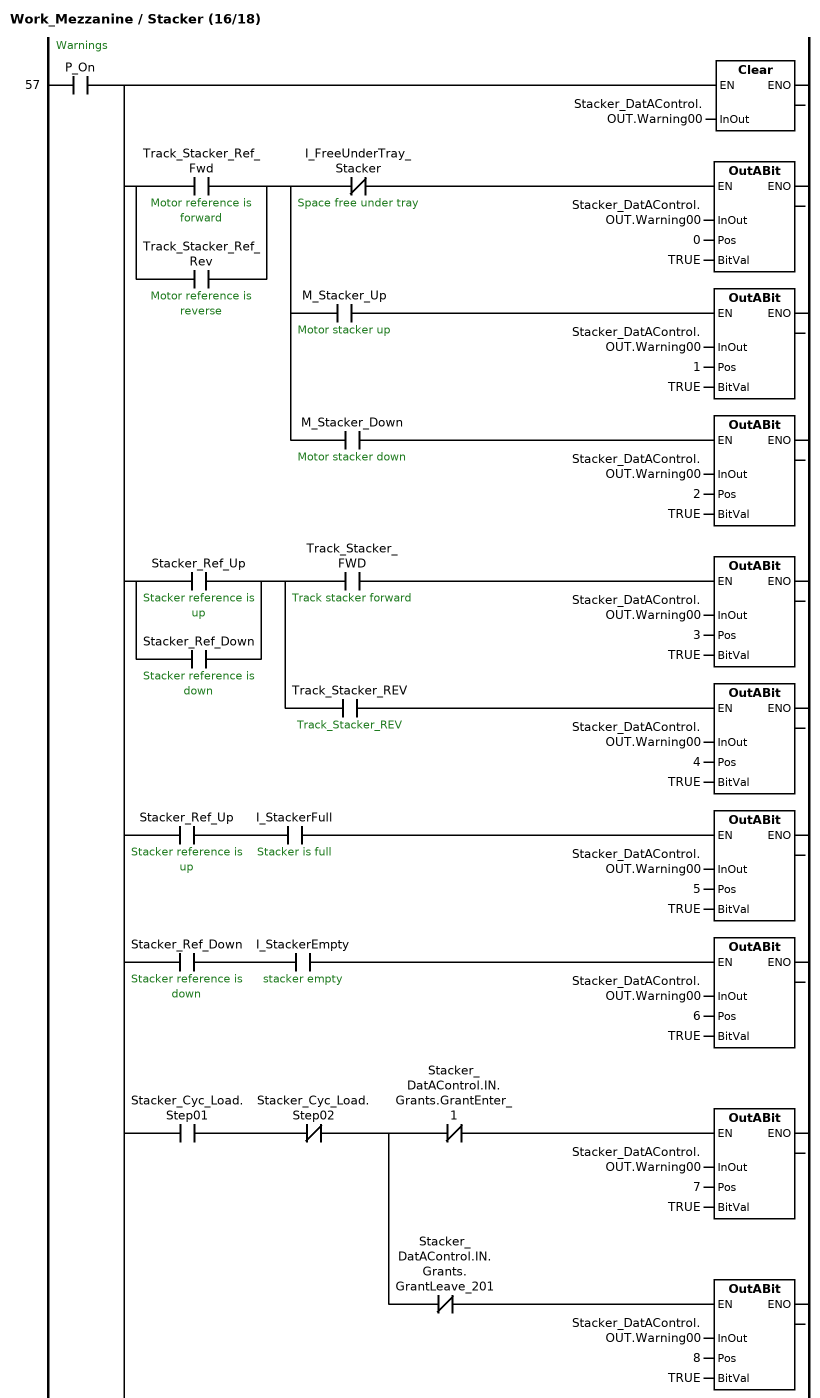
(* [picture p126: Work_Mezzanine / Stacker, rungs 57-57] *)

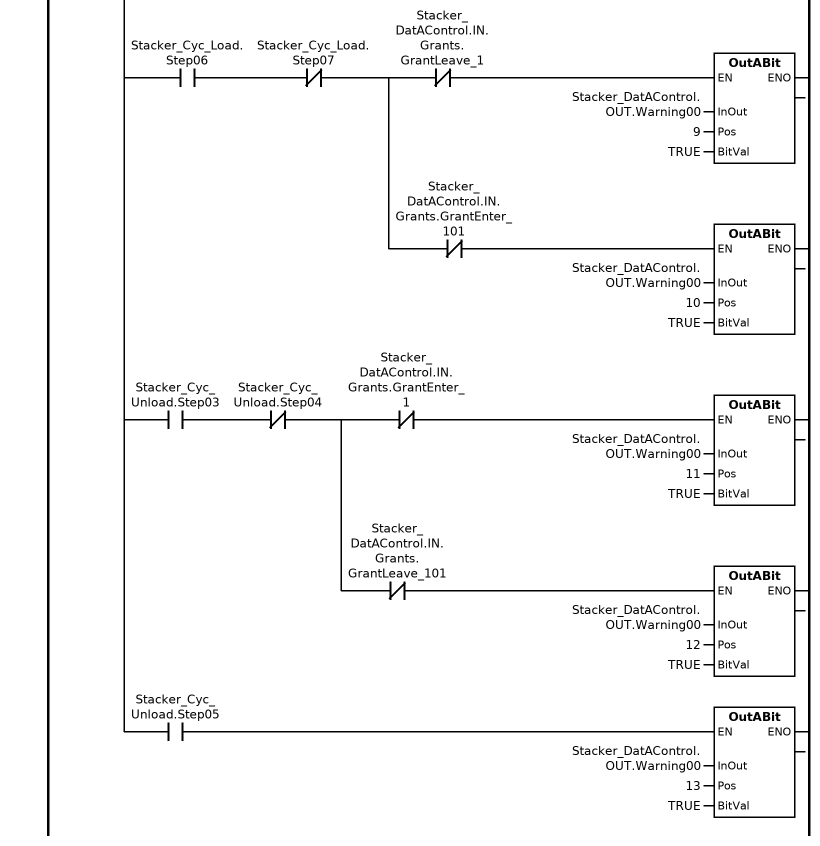
(* Rung 57: Warnings *)
IF P_On THEN Clear(InOut := Stacker_DatAControl.OUT.Warning00); END_IF;
_p6 := P_On AND (Track_Stacker_Ref_Fwd OR Track_Stacker_Ref_Rev);
IF _p6 AND NOT I_FreeUnderTray_Stacker THEN
    OutABit(InOut := Stacker_DatAControl.OUT.Warning00, Pos := 0, BitVal := TRUE);
END_IF;
IF _p6 AND M_Stacker_Up THEN
    OutABit(InOut := Stacker_DatAControl.OUT.Warning00, Pos := 1, BitVal := TRUE);
END_IF;
IF _p6 AND M_Stacker_Down THEN
    OutABit(InOut := Stacker_DatAControl.OUT.Warning00, Pos := 2, BitVal := TRUE);
END_IF;
IF P_On AND (Stacker_Ref_Up OR Stacker_Ref_Down) AND Track_Stacker_FWD THEN
    OutABit(InOut := Stacker_DatAControl.OUT.Warning00, Pos := 3, BitVal := TRUE);
END_IF;
IF P_On AND (Stacker_Ref_Up OR Stacker_Ref_Down) AND Track_Stacker_REV THEN
    OutABit(InOut := Stacker_DatAControl.OUT.Warning00, Pos := 4, BitVal := TRUE);
END_IF;
IF P_On AND Stacker_Ref_Up AND I_StackerFull THEN
    OutABit(InOut := Stacker_DatAControl.OUT.Warning00, Pos := 5, BitVal := TRUE);
END_IF;
IF P_On AND Stacker_Ref_Down AND I_StackerEmpty THEN
    OutABit(InOut := Stacker_DatAControl.OUT.Warning00, Pos := 6, BitVal := TRUE);
END_IF;
_p7 := P_On AND Stacker_Cyc_Load.Step01 AND NOT Stacker_Cyc_Load.Step02;
IF _p7 AND NOT Stacker_DatAControl.IN.Grants.GrantEnter_1 THEN
    OutABit(InOut := Stacker_DatAControl.OUT.Warning00, Pos := 7, BitVal := TRUE);
END_IF;
IF _p7 AND NOT Stacker_DatAControl.IN.Grants.GrantLeave_201 THEN
    OutABit(InOut := Stacker_DatAControl.OUT.Warning00, Pos := 8, BitVal := TRUE);
END_IF;
_p8 := P_On AND Stacker_Cyc_Load.Step06 AND NOT Stacker_Cyc_Load.Step07;
IF _p8 AND NOT Stacker_DatAControl.IN.Grants.GrantLeave_1 THEN
    OutABit(InOut := Stacker_DatAControl.OUT.Warning00, Pos := 9, BitVal := TRUE);
END_IF;
IF _p8 AND NOT Stacker_DatAControl.IN.Grants.GrantEnter_101 THEN
    OutABit(InOut := Stacker_DatAControl.OUT.Warning00, Pos := 10, BitVal := TRUE);
END_IF;
_p9 := P_On AND Stacker_Cyc_Unload.Step03 AND NOT Stacker_Cyc_Unload.Step04;
IF _p9 AND NOT Stacker_DatAControl.IN.Grants.GrantEnter_1 THEN
    OutABit(InOut := Stacker_DatAControl.OUT.Warning00, Pos := 11, BitVal := TRUE);
END_IF;
IF _p9 AND NOT Stacker_DatAControl.IN.Grants.GrantLeave_101 THEN
    OutABit(InOut := Stacker_DatAControl.OUT.Warning00, Pos := 12, BitVal := TRUE);
END_IF;
IF P_On AND Stacker_Cyc_Unload.Step05 THEN
    OutABit(InOut := Stacker_DatAControl.OUT.Warning00, Pos := 13, BitVal := TRUE);
END_IF;

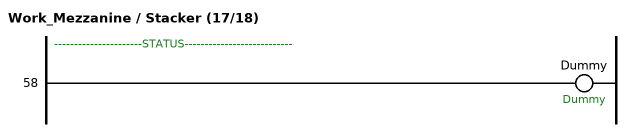
(* Rung 58: ----------------------STATUS--------------------------- *)
Dummy := TRUE;

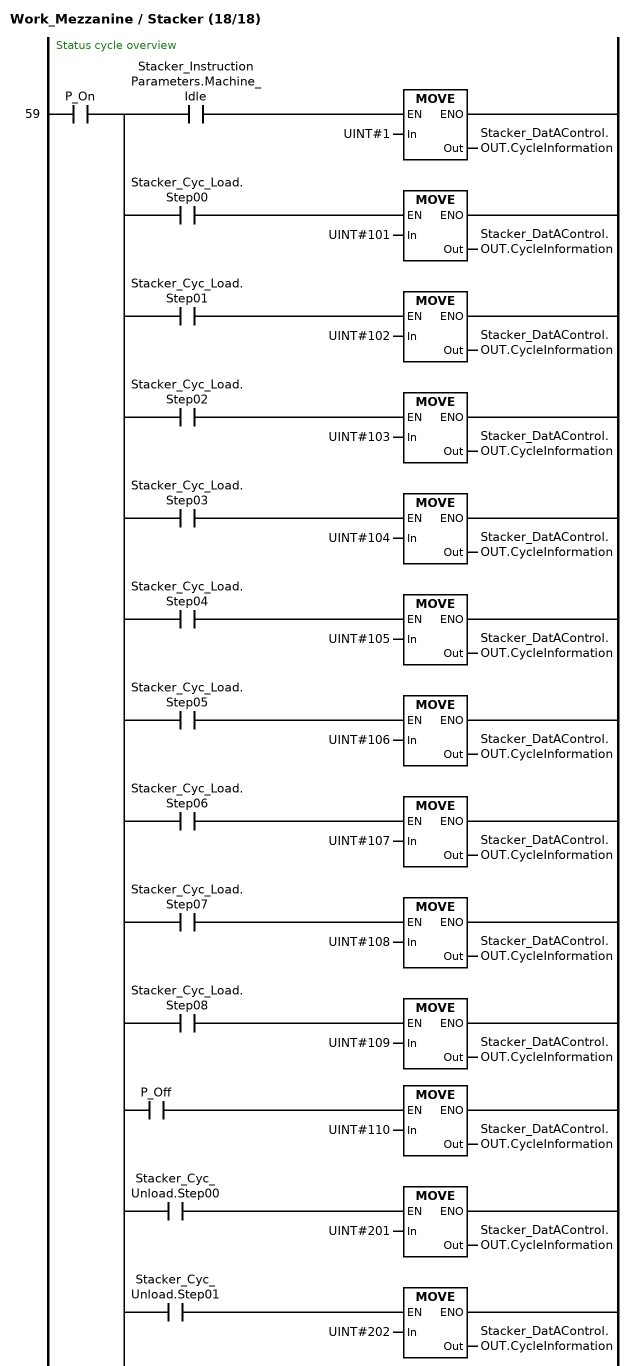

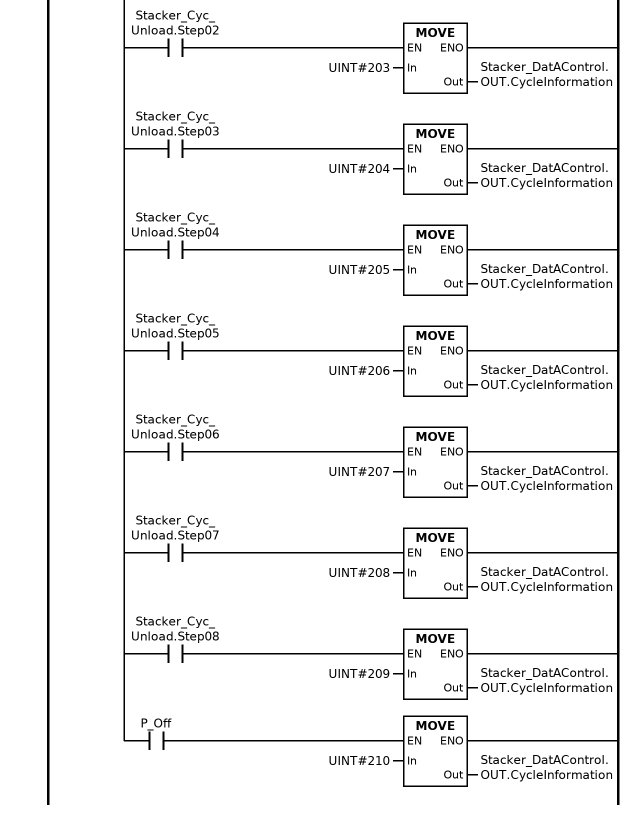
(* Rung 59: Status cycle overview *)
IF P_On AND Stacker_InstructionParameters.Machine_Idle THEN
    Stacker_DatAControl.OUT.CycleInformation := UINT#1;
END_IF;
IF P_On AND Stacker_Cyc_Load.Step00 THEN Stacker_DatAControl.OUT.CycleInformation := UINT#101; END_IF;
IF P_On AND Stacker_Cyc_Load.Step01 THEN Stacker_DatAControl.OUT.CycleInformation := UINT#102; END_IF;
IF P_On AND Stacker_Cyc_Load.Step02 THEN Stacker_DatAControl.OUT.CycleInformation := UINT#103; END_IF;
IF P_On AND Stacker_Cyc_Load.Step03 THEN Stacker_DatAControl.OUT.CycleInformation := UINT#104; END_IF;
IF P_On AND Stacker_Cyc_Load.Step04 THEN Stacker_DatAControl.OUT.CycleInformation := UINT#105; END_IF;
IF P_On AND Stacker_Cyc_Load.Step05 THEN Stacker_DatAControl.OUT.CycleInformation := UINT#106; END_IF;
IF P_On AND Stacker_Cyc_Load.Step06 THEN Stacker_DatAControl.OUT.CycleInformation := UINT#107; END_IF;
IF P_On AND Stacker_Cyc_Load.Step07 THEN Stacker_DatAControl.OUT.CycleInformation := UINT#108; END_IF;
IF P_On AND Stacker_Cyc_Load.Step08 THEN Stacker_DatAControl.OUT.CycleInformation := UINT#109; END_IF;
IF P_On AND P_Off THEN Stacker_DatAControl.OUT.CycleInformation := UINT#110; END_IF;
IF P_On AND Stacker_Cyc_Unload.Step00 THEN Stacker_DatAControl.OUT.CycleInformation := UINT#201; END_IF;
IF P_On AND Stacker_Cyc_Unload.Step01 THEN Stacker_DatAControl.OUT.CycleInformation := UINT#202; END_IF;
IF P_On AND Stacker_Cyc_Unload.Step02 THEN Stacker_DatAControl.OUT.CycleInformation := UINT#203; END_IF;
IF P_On AND Stacker_Cyc_Unload.Step03 THEN Stacker_DatAControl.OUT.CycleInformation := UINT#204; END_IF;
IF P_On AND Stacker_Cyc_Unload.Step04 THEN Stacker_DatAControl.OUT.CycleInformation := UINT#205; END_IF;
IF P_On AND Stacker_Cyc_Unload.Step05 THEN Stacker_DatAControl.OUT.CycleInformation := UINT#206; END_IF;
IF P_On AND Stacker_Cyc_Unload.Step06 THEN Stacker_DatAControl.OUT.CycleInformation := UINT#207; END_IF;
IF P_On AND Stacker_Cyc_Unload.Step07 THEN Stacker_DatAControl.OUT.CycleInformation := UINT#208; END_IF;
IF P_On AND Stacker_Cyc_Unload.Step08 THEN Stacker_DatAControl.OUT.CycleInformation := UINT#209; END_IF;
IF P_On AND P_Off THEN Stacker_DatAControl.OUT.CycleInformation := UINT#210; END_IF;
END_PROGRAM

PROGRAM ReadSettings
VAR_EXTERNAL
    Dummy : BOOL;
    Settings_CP : ST_Settings_CP;
    XTrack_X_Values : ARRAY[0..49] OF UDINT;
    XTrack_Y_Values : ARRAY[0..49] OF UDINT;
    Area : ARRAY[0..99] OF ST_Area;
    XTrack : ARRAY[0..49] OF ST_XTrack;
    Lift : ARRAY[0..9] OF ST_LiftInformation;
END_VAR
// Margins reservation system.
Settings_CP.Setting_Margin_X:= 1350; // Minimum margin = pallet 1200/2. 1270
Settings_CP.Setting_Margin_Y:= 700; // Minimum margin = Carrier lenght/2.

// Margin to define if carrier is in a certain area.
Settings_CP.Margin_AreaCompare:= 100;

// Values of position in X direction
XTrack_X_Values[0]:= 0;
XTrack_X_Values[1]:= 100000;
XTrack_X_Values[2]:= 102800;
XTrack_X_Values[3]:= 105600;
XTrack_X_Values[4]:= 108400;
XTrack_X_Values[5]:= 111516;
XTrack_X_Values[6]:= 114316;
XTrack_X_Values[7]:= 117116;
XTrack_X_Values[8]:= 119916;
XTrack_X_Values[9]:= 122716;
XTrack_X_Values[10]:= 125928;
XTrack_X_Values[11]:= 128728;
XTrack_X_Values[12]:= 131528;
XTrack_X_Values[13]:= 134328;
XTrack_X_Values[14]:= 137128;
XTrack_X_Values[15]:= 140244;
XTrack_X_Values[16]:= 143044;
XTrack_X_Values[17]:= 145844;
XTrack_X_Values[18]:= 148644;
XTrack_X_Values[19]:= 151444;

// Values of positions X-Track in Y direction
XTrack_Y_Values[0]:= 0;
XTrack_Y_Values[1]:= 100000;
XTrack_Y_Values[2]:= 108098;

// Dimensions of areas
// Check electrical lay-out for and overview of the Areas.

// This area is always 0
Area[0].Level:= 0;
Area[0].X_MIN:= 0;
Area[0].X_MAX:= 0;
Area[0].Y_Back:= 0;
Area[0].Y_Front:= 0;

// This is the 1st area on level 1, see lay-out for details.
// 1 to 9 = 100000 - 1/2 carrier with(650) to 122716 + 1/2 carrier with(650)
Area[11].Level:= 1;
Area[11].X_MIN:= 99350;
Area[11].X_MAX:= 123366;
Area[11].Y_Back:= 105198;
Area[11].Y_Front:= 110998;

// This is the 2nd area on level 1, see lay-out for details.
// 1 to 9
Area[12].Level:= 1;
Area[12].X_MIN:= 99350;
Area[12].X_MAX:= 123366;
Area[12].Y_Back:= 97100;
Area[12].Y_Front:= 102900; //carrier hit end @12981

// This is the 3th area on level 1, see lay-out for details.
// 10
Area[13].Level:= 1;
Area[13].X_MIN:= 125278;
Area[13].X_MAX:= 126578;
Area[13].Y_Back:= 98200;
Area[13].Y_Front:= 110998;

// This is the 4th area on level 1, see lay-out for details.
//1 to 19
Area[14].Level:= 1;
Area[14].X_MIN:= 128078;
Area[14].X_MAX:= 152094;
Area[14].Y_Back:= 105198;
Area[14].Y_Front:= 110998;

// This is the 5th area on level 1, see lay-out for details.
// 11 to 16
Area[15].Level:= 1;
Area[15].X_MIN:= 128078;
Area[15].X_MAX:= 143694;
Area[15].Y_Back:= 97100;
Area[15].Y_Front:= 102900;

// This is the 6th area on level 1, see lay-out for details.
// 17
Area[16].Level:= 1;
Area[16].X_MIN:= 145194;
Area[16].X_MAX:= 146494;
Area[16].Y_Back:= 98200;
Area[16].Y_Front:= 102900;

// This is the 7th area on level 1, see lay-out for details.
// 18 to 19
Area[17].Level:= 1;
Area[17].X_MIN:= 147994;
Area[17].X_MAX:= 152094;
Area[17].Y_Back:= 97100;
Area[17].Y_Front:= 102900;

// Copy areas to other levels
Area[21]:= Area[11];
Area[21].Level:= 2;
Area[31]:= Area[11];
Area[31].Level:= 3;
Area[41]:= Area[11];
Area[41].Level:= 4;
Area[51]:= Area[11];
Area[51].Level:= 5;
Area[61]:= Area[11];
Area[61].Level:= 6;
Area[71]:= Area[11];
Area[71].Level:= 7;

Area[22]:= Area[12];
Area[22].Level:= 2;
Area[32]:= Area[12];
Area[32].Level:= 3;
Area[42]:= Area[12];
Area[42].Level:= 4;
Area[52]:= Area[12];
Area[52].Level:= 5;
Area[62]:= Area[12];
Area[62].Level:= 6;
Area[72]:= Area[12];
Area[72].Level:= 7;

Area[23]:= Area[13];
Area[23].Level:= 2;
Area[33]:= Area[13];
Area[33].Level:= 3;
Area[43]:= Area[13];
Area[43].Level:= 4;
Area[53]:= Area[13];
Area[53].Level:= 5;
Area[63]:= Area[13];
Area[63].Level:= 6;
Area[73]:= Area[13];
Area[73].Level:= 7;

Area[24]:= Area[14];
Area[24].Level:= 2;
Area[34]:= Area[14];
Area[34].Level:= 3;
Area[44]:= Area[14];
Area[44].Level:= 4;
Area[54]:= Area[14];
Area[54].Level:= 5;
Area[64]:= Area[14];
Area[64].Level:= 6;
Area[74]:= Area[14];
Area[74].Level:= 7;

Area[25]:= Area[15];
Area[25].Level:= 2;
Area[35]:= Area[15];
Area[35].Level:= 3;
Area[45]:= Area[15];
Area[45].Level:= 4;
Area[55]:= Area[15];
Area[55].Level:= 5;
Area[65]:= Area[15];
Area[65].Level:= 6;
Area[75]:= Area[15];
Area[75].Level:= 7;

Area[26]:= Area[16];
Area[26].Level:= 2;
Area[36]:= Area[16];
Area[36].Level:= 3;
Area[46]:= Area[16];
Area[46].Level:= 4;
Area[56]:= Area[16];
Area[56].Level:= 5;
Area[66]:= Area[16];
Area[66].Level:= 6;
Area[76]:= Area[16];
Area[76].Level:= 7;

Area[27]:= Area[17];
Area[27].Level:= 2;
Area[37]:= Area[17];
Area[37].Level:= 3;
Area[47]:= Area[17];
Area[47].Level:= 4;
Area[57]:= Area[17];
Area[57].Level:= 5;
Area[67]:= Area[17];
Area[67].Level:= 6;
Area[77]:= Area[17];
Area[77].Level:= 7;

 // Information about X-Tracks
XTrack[0].XTrack_Number:= 0;
XTrack[0].MinimumPosition:= 0;
XTrack[0].MaximumPosition:= 0;
	 
XTrack[1].XTrack_Number:= 1;
XTrack[1].MinimumPosition:= 1;
XTrack[1].MaximumPosition:= 19;

XTrack[2].XTrack_Number:= 2;
XTrack[2].MinimumPosition:= 1;
XTrack[2].MaximumPosition:= 19;

// Information about lifts
// This lift is always 0
Lift[0].Number:= 0;
Lift[0].X_Coordinate_Lift_MIN:= 0;
Lift[0].X_Coordinate_Lift_MAX:= 0;
Lift[0].Y_Coordinate_Lift_Back:= 0;
Lift[0].Y_Coordinate_Lift_Front:= 0;
Lift[0].Y_Coordinate_LiftCenter:= 0;
Lift[0].Pos_Lift_XTrack:= FALSE;

// This is the lift in growing room3
Lift[1].Number:= 1;
Lift[1].X_Coordinate_Lift_MIN:= 125278;
Lift[1].X_Coordinate_Lift_MAX:= 126578;
Lift[1].Y_Coordinate_Lift_Back:= 98100;
Lift[1].Y_Coordinate_Lift_Front:= 99390;
Lift[1].Y_Coordinate_LiftCenter:= 98223; 
Lift[1].Pos_Lift_XTrack:= FALSE;

// This is the lift in growing room4 ;
Lift[2].Number:= 2;
Lift[2].X_Coordinate_Lift_MIN:= 145194;
Lift[2].X_Coordinate_Lift_MAX:= 146494;
Lift[2].Y_Coordinate_Lift_Back:= 98100;
Lift[2].Y_Coordinate_Lift_Front:= 99390;
Lift[2].Y_Coordinate_LiftCenter:= 98223;
Lift[2].Pos_Lift_XTrack:= FALSE;
END_PROGRAM

FUNCTION PositionResetCheck : BOOL
VAR_INPUT
    Level : UINT;  (* Level *)
    X_Track : UINT;  (* X-Track *)
    Position : UINT;  (* Position *)
END_VAR
(* ladder, written here as Structured Text *)

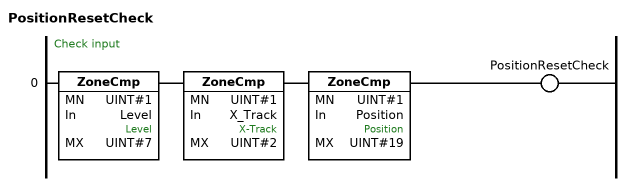
(* Rung 0: Check input *)
PositionResetCheck := ZoneCmp(MN := UINT#1, In := Level, MX := UINT#7) AND ZoneCmp(MN := UINT#1, In := X_Track, MX := UINT#2) AND ZoneCmp(MN := UINT#1, In := Position, MX := UINT#19);
END_FUNCTION

FUNCTION PositionInformationRack : BOOL
VAR
    Counter : UINT;  (* Counter FOR loop *)
END_VAR
VAR_INPUT
    X : UDINT;  (* Actual X position *)
    Y : UDINT;  (* Actual Y position *)
    Z : UDINT;  (* Actual Z position *)
    Margin : UDINT;  (* Margin for area compare *)
    Areas : ARRAY[0..99] OF ST_Area;
END_VAR
VAR_OUTPUT
    O_Area : ST_Area;  (* Area where carrier is in *)
END_VAR
Clear(O_Area);

FOR Counter := 0 TO 99 BY 1 DO
	IF Z = Areas[Counter].Level AND
		X >= (Areas[Counter].X_MIN - Margin) AND
		X <= (Areas[Counter].X_MAX + Margin) AND
		Y >= (Areas[Counter].Y_Back - Margin) AND
		Y <= (Areas[Counter].Y_Front + Margin) THEN
		O_Area := Areas[Counter];
		EXIT;
	END_IF;
END_FOR;
END_FUNCTION

FUNCTION PositionInformationXTrack : BOOL
VAR
    Counter : UINT;
END_VAR
VAR_INPUT
    Y : UDINT;  (* Actual Y position *)
    XTrack_Y_Values : ARRAY[0..49] OF UDINT;  (* X-Track Y values *)
END_VAR
VAR_OUTPUT
    X_Track_Number : UINT;  (* Matchin X-Track number *)
END_VAR
X_Track_Number := 0;

FOR Counter := 0 TO 49 BY 1 DO
    IF XTrack_Y_Values[Counter] >= (Y - 20) AND
		XTrack_Y_Values[Counter] <= (Y + 20) THEN
		X_Track_Number := Counter;
		EXIT;
	END_IF;
END_FOR;
END_FUNCTION

FUNCTION DefineTransferGate : BOOL
VAR
    Counter : UINT;  (* Counter FOR loop *)
END_VAR
VAR_INPUT
    X : UDINT;  (* Actual X position *)
    Y : UDINT;  (* Actual Y position *)
    Z : UDINT;  (* Actual Z position *)
    XTrack_X_Values : ARRAY[0..49] OF UDINT;  (* X Track X values *)
END_VAR
VAR_OUTPUT
    Transfergate : UINT;  (* Transfergate *)
END_VAR
Transfergate := 0;

IF (Z <> 0 AND Y <> 0 AND X <> 0) THEN
	// Z value
	Transfergate := UDINT_TO_UINT(Z) * 1000;

	// Y value
	// Section A
	IF Y > 108098 THEN
		Transfergate := Transfergate + 300;
	// Section B
	ELSIF Y < 108098 AND Y > 104216 THEN
		Transfergate:= Transfergate + 200;
	// Section C
	ELSIF Y < 104216 AND Y > 100000 THEN
		Transfergate:= Transfergate + 100;
	// Section D
	ELSIF Y < 10000 THEN
		Transfergate:= Transfergate + 0;	
	END_IF;

	// X value
	FOR Counter := 0 TO 49 BY 1 DO
		IF X = XTrack_X_Values[Counter] THEN
			Transfergate := Transfergate + Counter;
			EXIT;
		END_IF;
	END_FOR;
END_IF;
END_FUNCTION

FUNCTION_BLOCK FB_40401
VAR
    NOP : BOOL;  (* NOP *)
    Dummy : BOOL;  (* Dummy *)
    LS_FallProtect : FB_101;
    I_LS_Fallprotect : BOOL;  (* Limit switch fall protection *)
    LS_Lift_Up : FB_101;
    I_LS_Lift_Up : BOOL;  (* Limit switch lift up *)
    LS_Lift_Down : FB_101;
    I_LS_Lift_Down : BOOL;  (* Limit switch lift down *)
    LC_Car_Free_Back : FB_101;
    I_LC_Car_Free_Back : BOOL;  (* Photocell carrier detection free backside *)
    LC_Car_Present : FB_101;
    I_LC_Car_Present : BOOL;  (* Photocell carrier present *)
    LC_Car_Free_Front : FB_101;
    I_LC_Car_Free_Front : BOOL;  (* Photocell carrier detection free frontside *)
    LC_Con_Free_Back : FB_101;
    I_LC_Con_Free_Back : BOOL;  (* Photocell container detection free backside *)
    LC_Con_Present : FB_101;
    I_LC_Con_Present : BOOL;  (* Photocell container present *)
    LC_Con_Free_Front : FB_101;
    I_LC_Con_Free_Front : BOOL;  (* Photocell container detection free frontside *)
    IS_Act_Back_Out : FB_101;
    I_IS_Act_Back_Out : BOOL;  (* Inductive sensor actuator backside out *)
    IS_Act_Back_In : FB_101;
    I_IS_Act_Back_In : BOOL;  (* Inductive sensor actuator backside in *)
    IS_Act_Front_Out : FB_101;
    I_IS_Act_Front_Out : BOOL;  (* Inductive sensor actuator frontside out *)
    IS_Act_Front_In : FB_101;
    I_IS_Act_Front_In : BOOL;  (* Inductive sensor actuator frontside in *)
    IS_Lift_Level : FB_101;
    I_IS_Lift_Level : BOOL;  (* Inductive sensor lift at a level *)
    InstructionLift : FB_902;
    ConditionsLiftOk : BOOL;  (* Conditions move lift Ok *)
    Lift : FB_203;
    ConditionsLiftUpOK : BOOL;  (* Conditions move lift up OK *)
    ConditionsLiftDownOK : BOOL;  (* Conditions move lift down OK *)
    LiftMotorUp : BOOL;  (* Lift motor up *)
    LiftMotorDown : BOOL;
    LiftGoLowSpeed : BOOL;  (* Lift go low speed *)
    LiftMotorReversal : FB_201;
    O_LiftMotorUp : BOOL;  (* Lift motor up *)
    O_LiftMotorDown : BOOL;  (* Lift motor down *)
    T_Reversal_Lift : BOOL;  (* Timer reversal protection *)
    InstructionParameterIn : ST_FB_009xx\FB_902_ParametersIN;  (* Instruction parameter in *)
    InstructionParameterOut : ST_FB_009xx\FB_902_ParametersOUT;  (* Instruction parameter out *)
    LiftDesiredUp_Auto : BOOL;  (* Lift desired up in automatic *)
    LiftDesiredUp_Manual : BOOL;  (* Lift desired up in manual *)
    LiftDesiredDown_Auto : BOOL;  (* Lift desired down in automatic *)
    LiftDesiredDown_Manual : BOOL;  (* Lift desired down in manual *)
    ManualControl_Lift : FB_303;
    Des_Speed_Lift : UINT;  (* Desired speed lift *)
    AtPositionLift : BOOL;  (* Lift is at position *)
    ActuatorFront : FB_1002;
    CounterActuatorFront : UDINT;  (* Counter total movements actuator front *)
    ActuatorBack : FB_1002;
    CounterActuatorBack : UDINT;  (* Counter total movements actuator back *)
    O_ChainFWD : BOOL;  (* Chain motor forward *)
    O_ChainREV : BOOL;  (* Chain motor reverse *)
    Des_Speed_Chain : UINT;  (* Desired speed chain *)
    Write_Param_Lift : BOOL;
    Read_Param_Lift : BOOL;
    Write_Param_Chain : BOOL;
    Read_Param_Chain : BOOL;
END_VAR
VAR RETAIN
    LiftLoaded : BOOL;  (* Status lift is loaded (1 = loaded 0= not loaded) *)
END_VAR
VAR
    MachineInAlarm : BOOL;  (* Machine is in alarm *)
END_VAR
VAR RETAIN
    Cyc_Mov : ST_FB_40401_Cyc_Move;  (* Cycle move *)
    Cyc_LoadBench : ST_FB_40401_Cyc_LoadBench;  (* Cycle load bench *)
    Cyc_UnloadBench : ST_FB_40401_Cyc_UnloadBench;  (* Cycle unload bench *)
    Cyc_LoadCarrier : ST_FB_40401_Cyc_LoadCarrier;  (* Cycle load carrier *)
    Cyc_UnloadCarrier : ST_FB_40401_Cyc_UnloadCarrier;  (* Cycle unload carrier *)
    Cyc_Attach : ST_FB_40401_Cyc_Attach;  (* Cycle attach; Step00 Attach is desired, move actuator out (Stopper down) *)
    Cyc_Detach : ST_FB_40401_Cyc_Detach;  (* Cycle detach; Step00 Attach is desired, move actuators in (Stoppers up) *)
END_VAR
VAR
    NoInstructionActive : BOOL;  (* No instruction active *)
    Con_Actuator_Ok : BOOL;  (* Condition lift actuator okay *)
    Con_Sensor_Carrier : BOOL;  (* Condition lift sensor detecting carrier okay *)
    Con_Sensor_Move : BOOL;  (* Condition lift sensors okay *)
    Con_Lift_Free : BOOL;  (* Condition lift sensor free backside/frontside *)
    Con_Sensor_Bench : BOOL;  (* Condition lift sensor bench *)
    ConditionStart : BOOL;  (* Start conditions lift OK *)
    T_LiftAtPosition : _sTimer;  (* Timer lift at position *)
END_VAR
VAR RETAIN
    CarrierLoaded : BOOL;  (* Status carrier loaded *)
END_VAR
VAR
    PositionReference : UDINT;  (* Position reference intern *)
    Act_Front_Cur_Pos : UDINT;  (* Actuator frontside current position *)
    Act_Back_Ref_Pos : UDINT;  (* Actuator backside reference position *)
    Act_Front_Ref_Pos : UDINT;  (* Actuator frontside reference position *)
    Act_Back_Cur_Pos : UDINT;  (* Actuator backside current position *)
    DOff_LC_Con_Free_front : BOOL;  (* Delay off photocell carrier detection free frontside *)
    DOff_LC_Con_Free_Back : BOOL;  (* Delay off photocell container detection free backside *)
    DON_LC_Con_Free_front : BOOL;  (* Delay on photocell carrier detection free frontside *)
    DON_LC_Con_Free_Back : BOOL;  (* Delay on photocell container detection free backside *)
    TransferOK : BOOL;  (* Transfer is OK *)
    T_LiftEmpty : _sTimer;  (* Timer lift is empty *)
    ConditionsChainOk : BOOL;  (* Global conditions chain conveyer ok *)
    ConditionsChainFWD : BOOL;  (* Conditions chain conveyer forward ok *)
    ConditionsChainREV : BOOL;  (* Conditions chain conveyer backward ok *)
    ChainDesiredFWD_Auto : BOOL;  (* Chain conveyer desired forward in automatic *)
    ChainDesiredREV_Auto : BOOL;  (* Chain conveyer desired backward in automatic *)
    ManualControl_Chain : FB_303;
    ChainDesiredFWD_Manual : BOOL;  (* Chain conveyer desired forward in manual *)
    ChainDesiredREV_Manual : BOOL;  (* Chain conveyer desired reverse in manual *)
    ChainConveyer : FB_203;
    ChainMotorFWD : BOOL;  (* Chain conveyer motor forward *)
    ChainMotorREV : BOOL;  (* Chain conveyer motor reverse *)
    ChainMotorReversal : FB_201;
    T_Reversal_Chain : BOOL;  (* Reversal timer chain converyer *)
    TimerChainSlow : _sTimer;  (* Timer chain slow speed *)
    MachineMode : ST_MachineMode;  (* Machine mode *)
    ModuloRemainder1000 : UINT;  (* Remainder 1000 *)
    ModuloRemainder100 : UINT;  (* Remainder 100s *)
    InstructionSideFront : BOOL;  (* Instruction side is front *)
    InstructionSideBack : BOOL;  (* Instruction side is back *)
    Current_Position : UINT;  (* Current position of lift (MachineLocation) *)
    index : UINT;  (* Index for position calculation *)
    FB_Inverter_Lift : FB_305;
    FB_Inverter_Chain : FB_305;
    PositionReference_LowMargin : UDINT;  (* Lower margine prosition reference *)
    PositionReference_HighMargin : UDINT;  (* Higher margine prosition reference *)
    NeedLevelSensor : BOOL;  (* Position needs level sensor *)
END_VAR
VAR RETAIN
    EncoderLiftOvershootUp : UDINT;
    EncoderLiftOvershootDown : UDINT;
END_VAR
VAR
    EncoderLiftAtPosition : UDINT;
    Overshoot_Position : UINT;
    AtPositionLiftNotMoving : BOOL;
    DON_LC_Car_Free_Back : BOOL;  (* Delay on photocell carrier detection free backside *)
    DON_LC_Car_Present : BOOL;  (* Delay on photocell carrier present *)
    DON_LC_Car_Free_Front : BOOL;  (* Delay on photocell carrier detection free frontside *)
    DON_LC_Con_Present : BOOL;  (* Delay on photocell container present *)
    TimerStopperfront_Notup : _sTimer;  (* Timer stopper frontside not up *)
    TimerStopperFront_StillUp : _sTimer;  (* Timer stopper frontside is still up *)
    TimerStopperBack_Notup : _sTimer;  (* Timer stopper Backside not up *)
    TimerStopperBack_StillUp : _sTimer;  (* Timer stopper backside is still up *)
    Traystopper_F_Manual_Up : BOOL;  (* Traystopper manual up *)
    Traystopper_B_Manual_Up : BOOL;  (* Traystopper manual up *)
    TimerConditionsNotOk : _sTimer;  (* Timer conditions not OK *)
    IS_Con_In_Pos_Back : FB_101;
    I_IS_Con_In_Pos_Back : BOOL;  (* Inductive sensor tray in position back *)
    DON_IS_Con_In_Pos_Back : BOOL;  (* inductive sensor tray is in position back delay on *)
    DOFF_IS_Con_In_Pos_Back : BOOL;  (* Inductive sensor tray is in position back delay off *)
    IS_Con_In_Pos_Front : FB_101;
    I_IS_Con_In_Pos_Front : BOOL;  (* Inductive sensor tray is in position front *)
    DON_IS_Con_In_Pos_Front : BOOL;  (* Inductive sensor tray is in position front delay on *)
    DOFF_IS_Con_In_Pos_Front : BOOL;  (* Inductive sensor tray is in position front delay off *)
    T_AttachDone : _sTimer;  (* This timer make sure the new carrier position is red by DAC *)
    ConditionsActuatorFrontOk : BOOL;  (* Global conditions actuator front ok *)
    ConditionsActuatorBackOk : BOOL;  (* Global conditions actuator back ok *)
    Lift_Direction : BOOL;  (* Lift direction 0=down, 1= up *)
    LiftDesiredUp : BOOL;
    LiftDesiredDown : BOOL;
    LiftDirectionUp : BOOL;
    LiftDirectionDown : BOOL;
    T_AtPositionNotOk : _sTimer;  (* Timer at position not OK *)
    T_MachineInAlarm : _sTimer;
    AlarmEncoderNoPulses : BOOL;
    AlarmEncoderDirection : BOOL;
    Alarm_NoPulses : FB_504;
    LiftStuck : BOOL;
    Alarm_WrongDirection : FB_503;
    Lif : BOOL;
    Lift_Free_Back : FB_311;
    Lift_Free_Back_OK : BOOL;  (* Sensor lift free back OK *)
    Lift_Free_Front : FB_311;
    Lift_Free_Front_OK : BOOL;  (* Sensor lift free front OK *)
    PositionReference_LowMargin_Warning : UDINT;
    PositionReference_HighMargin_Warning : UDINT;
    Warning_AtPositionLift : BOOL;
    ConditionStartMove : BOOL;  (* Start conditions move cyce OK *)
    LastMobileMachineTalkedTo : UINT;  (* Remember what the last machine was lift talked to. *)
    LastMachineCycle : UINT;  (* Last machine cycl *)
    T_Instr_Too_Long : _sTimer;  (* Timer instruction is too lon *)
    MinimumPosition : UDINT;
    ResetValueUpper : UDINT;
    ResetValueLower : UDINT;
    PositionToResetOK : BOOL;  (* Lift position is within the margin to reset *)
END_VAR
VAR_INPUT
    Enable : BOOL;  (* Enable *)
    EmergencystopOk : BOOL;  (* emergency stop is OK *)
    Inputs : ST_FB_40401_InputsLift;
    EncoderLift : UDINT;  (* Encoder value lift *)
    Settings : ST_FB_40401_SettingsLift;  (* MinimumSpeed Setting: Minimum speed; SafeStopTime Setting safe stop time; Dec_Area_High Setting: Decelerate area high value (where deceleration begins); Dec_Area_Low Setting: Decelerate area low value (where deceleration ends); MaximumSpeed Setting: Maximum speed; MinimumPulseLevel Setting: Minimum pulse level; MaximumPulseLevel Setting: Maximum pulse level; ActuatorsLastPosition Actuator can stay in the last position; ActuatorBackOn Actuator backside on; ActuatorFrontOn Actuator frontside on; PositionReferenceOk Setting position referece is Ok; LoadGateOk Setting load gate is Ok; UnloadGateOk Setting unload gate is Ok; ChainHighSpeed Setting chain conveyer high speed; UseBenchUnloadInstruction Use unload instruction; UnloadToLOcation Unload to location; TimeConFreeFrontDOFF Time delay off; TimeConFreeFrontDON Time delay on; TimeConFreeBackDON Time delay on; TimeConFreeBackDOFF Time delay off; TimeConInductiveBackDON Setting time delay on; TimeConInductiveBackDOFF Setting time delay off; TimeConInductiveFrontDON Setting time delay on; TimeConInductiveFrontDOFF Setting time delay off; Option_InductiveTraydetection Option use Inductive sensors *)
    UserSettings : ST_FB_40401_UserSetting;  (* Overrule_LC_Front User overrule LC front; Overrule_LC_Back User overrule LC back *)
    MX2StatusLift : ST_MX2\Status;
    MX2StatusChain : ST_MX2\Status;
    InverterSpeed : UINT;  (* Inverter speed in hz *)
    CarrierCommIn : ST_Comm_MobileMachine_To_Lift;
    FrontCommIn : ST_FB_40401_CommIn;  (* RequestSignal Request signal *)
    BackCommIn : ST_FB_40401_CommIn;  (* RequestSignal request signal *)
END_VAR
VAR_OUTPUT
    Outputs : ST_FB_40401_OutputsLift;
    ResetEncoder : BOOL;
    ResetValue : UDINT;
    MX2CommandLift : ST_MX2\Command;
    MX2SpeedRefLift : UINT;
    MX2CommandChain : ST_MX2\Command;
    MX2SpeedRefChain : UINT;
    CarrierCommOut : ST_Comm_Lift_To_MobileMachine;
    FrontCommOut : ST_FB_40401_CommOut;  (* SupplySignal Supply signal ; RequestSignal Request signal; StopOutbound Stop outbound *)
    BackCommOut : ST_FB_40401_CommOut;  (* SupplySignal Supply signal; RequestSignal request signal; StopOutbound Stop outbound *)
    Extra_Warning1 : WORD;  (* Extra warning 1 *)
    Extra_Warning2 : WORD;  (* Extra warning 2 *)
    Extra_Warning3 : WORD;  (* Extra warning 3 *)
    Status : ST_FB_40401_Status;  (* Lift_With_Bench Status loaded with bench; Lift_With_Loaded_Carrier Status lift with loaded carrier; Lift_With_Unloaded_Carrier Status lift with unloaded carrier *)
END_VAR
VAR_IN_OUT
    DatAControl : ST_DatAControl_Standard;  (* IN.MachineMode Machine mode; IN Data control in; OUT Dat A Control out; IN.Instruction.Operand1 Operand 1; IN.Settings.ResetAlarm Reset alar *)
    Commands : ST_FB_40401_Commands;  (* TraystopperFront Commands traystopper; TraystopperBack Commands traystopper *)
    TransferBuffer : ST_TransferBuffer;  (* Transfer buffer *)
END_VAR
VAR_EXTERNAL
    DatAControl_Lift04 : ST_DatAControl_Standard;
    ES_OK : BOOL;
    EncoderLift03 : UDINT;
    DatAControl_Lift03 : ST_DatAControl_Standard;
END_VAR
VAR
    _t1 : BOOL;
    _e2 : R_TRIG;
    _t3 : BOOL;
    _p4 : BOOL;
    _p5 : BOOL;
    _e6 : R_TRIG;
    _e7 : R_TRIG;
    _e8 : R_TRIG;
    _e9 : R_TRIG;
    _e10 : R_TRIG;
    _e11 : R_TRIG;
    _p12 : BOOL;
    _t13 : BOOL;
    _e14 : R_TRIG;
    _e15 : R_TRIG;
    _p16 : BOOL;
    _e17 : R_TRIG;
    _p18 : BOOL;
    _e19 : R_TRIG;
    _e20 : R_TRIG;
    _p21 : BOOL;
    _t22 : BOOL;
    _e23 : R_TRIG;
    _e24 : R_TRIG;
    _e25 : R_TRIG;
    _e26 : R_TRIG;
    _e27 : R_TRIG;
    _e28 : R_TRIG;
    _e29 : R_TRIG;
    _e30 : R_TRIG;
    _e31 : R_TRIG;
    _e32 : R_TRIG;
    _e33 : R_TRIG;
    _e34 : R_TRIG;
    _e35 : R_TRIG;
    _e36 : R_TRIG;
    _e37 : R_TRIG;
    _e38 : R_TRIG;
    _e39 : R_TRIG;
    _e40 : R_TRIG;
    _e41 : R_TRIG;
    _e42 : R_TRIG;
    _p43 : BOOL;
    _p44 : BOOL;
    _p45 : BOOL;
    _p46 : BOOL;
    _p47 : BOOL;
    _e48 : R_TRIG;
    _e49 : F_TRIG;
    _p50 : BOOL;
    _e51 : R_TRIG;
    _p52 : BOOL;
    _p53 : BOOL;
    _t54 : BOOL;
    _p55 : BOOL;
    _t56 : BOOL;
    _e57 : R_TRIG;
    _e58 : R_TRIG;
    _e59 : R_TRIG;
    _e60 : R_TRIG;
    _e61 : R_TRIG;
    _t62 : BOOL;
    _t63 : BOOL;
    _e64 : R_TRIG;
    _e65 : R_TRIG;
    _t66 : BOOL;
    _t67 : BOOL;
    _t68 : BOOL;
    _br447_0 : BOOL;
    _br447_1 : BOOL;
    _br447_2 : BOOL;
    _br447_3 : BOOL;
    _br447_4 : BOOL;
    _t69 : BOOL;
    _e70 : R_TRIG;
    _t71 : BOOL;
    _t72 : BOOL;
    _p73 : BOOL;
    _e74 : R_TRIG;
    _e75 : R_TRIG;
    _e76 : R_TRIG;
END_VAR
(* ladder, written here as Structured Text *)

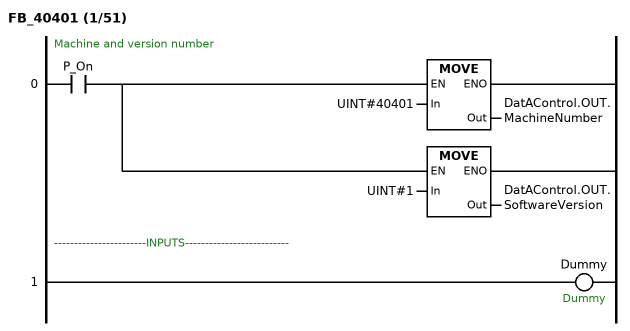
(* Rung 0: Machine and version number *)
IF P_On THEN
    DatAControl.OUT.MachineNumber := UINT#40401;
    DatAControl.OUT.SoftwareVersion := UINT#1;
END_IF;
(* Rung 1: -----------------------INPUTS-------------------------- *)
Dummy := TRUE;

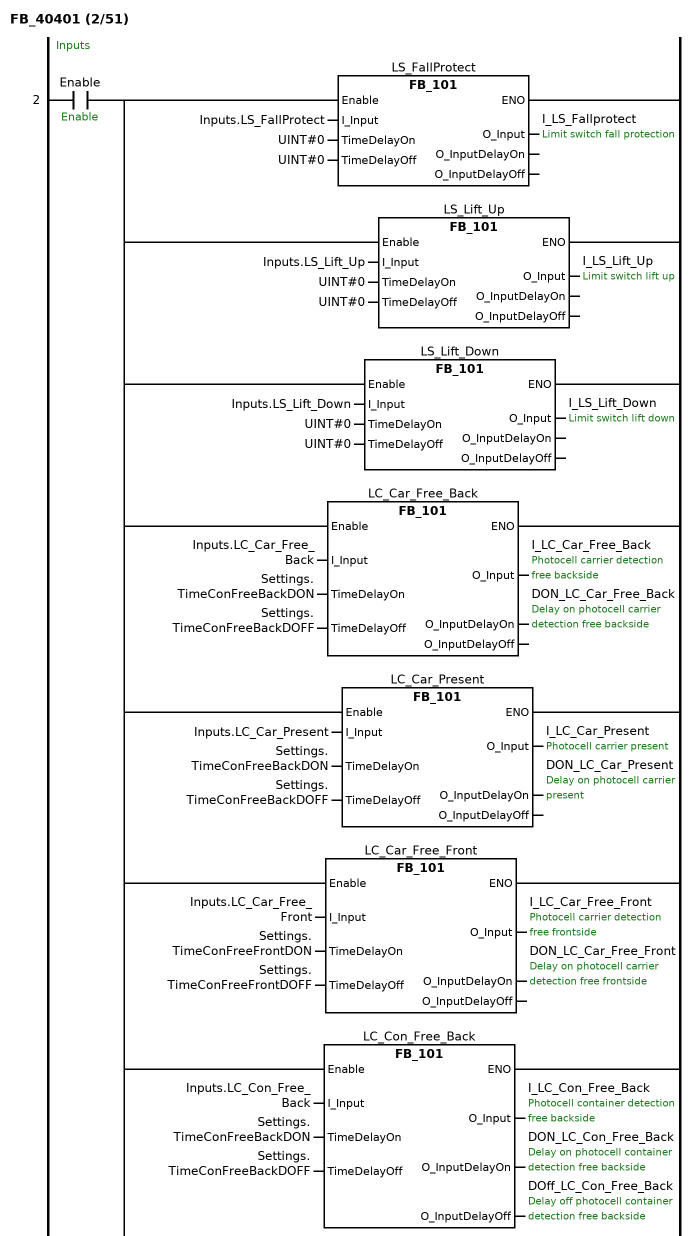

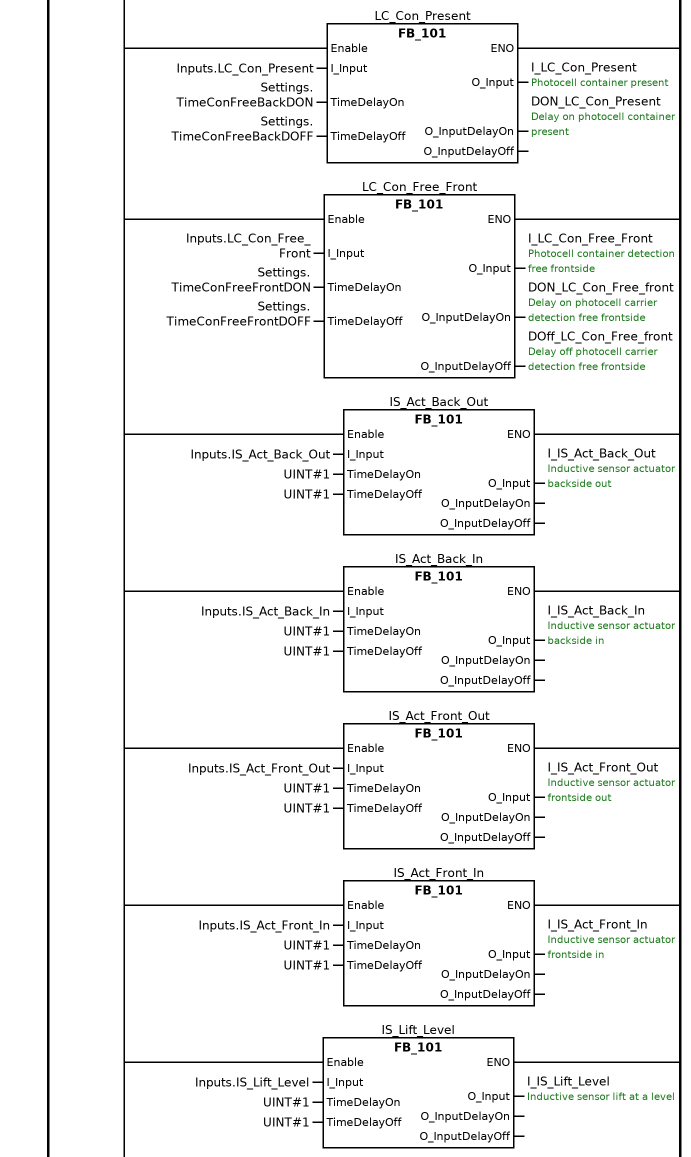

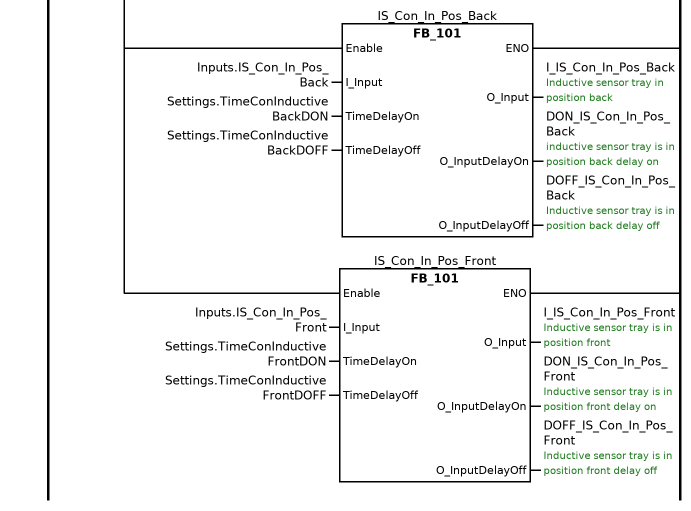
(* Rung 2: Inputs *)
LS_FallProtect(Enable := Enable, I_Input := Inputs.LS_FallProtect, TimeDelayOn := UINT#0, TimeDelayOff := UINT#0, O_Input => I_LS_Fallprotect);
LS_Lift_Up(Enable := Enable, I_Input := Inputs.LS_Lift_Up, TimeDelayOn := UINT#0, TimeDelayOff := UINT#0, O_Input => I_LS_Lift_Up);
LS_Lift_Down(Enable := Enable, I_Input := Inputs.LS_Lift_Down, TimeDelayOn := UINT#0, TimeDelayOff := UINT#0, O_Input => I_LS_Lift_Down);
LC_Car_Free_Back(Enable := Enable, I_Input := Inputs.LC_Car_Free_Back, TimeDelayOn := Settings.TimeConFreeBackDON, TimeDelayOff := Settings.TimeConFreeBackDOFF, O_Input => I_LC_Car_Free_Back, O_InputDelayOn => DON_LC_Car_Free_Back);
LC_Car_Present(Enable := Enable, I_Input := Inputs.LC_Car_Present, TimeDelayOn := Settings.TimeConFreeBackDON, TimeDelayOff := Settings.TimeConFreeBackDOFF, O_Input => I_LC_Car_Present, O_InputDelayOn => DON_LC_Car_Present);
LC_Car_Free_Front(Enable := Enable, I_Input := Inputs.LC_Car_Free_Front, TimeDelayOn := Settings.TimeConFreeFrontDON, TimeDelayOff := Settings.TimeConFreeFrontDOFF, O_Input => I_LC_Car_Free_Front, O_InputDelayOn => DON_LC_Car_Free_Front);
LC_Con_Free_Back(Enable := Enable, I_Input := Inputs.LC_Con_Free_Back, TimeDelayOn := Settings.TimeConFreeBackDON, TimeDelayOff := Settings.TimeConFreeBackDOFF, O_Input => I_LC_Con_Free_Back, O_InputDelayOn => DON_LC_Con_Free_Back, O_InputDelayOff => DOff_LC_Con_Free_Back);
LC_Con_Present(Enable := Enable, I_Input := Inputs.LC_Con_Present, TimeDelayOn := Settings.TimeConFreeBackDON, TimeDelayOff := Settings.TimeConFreeBackDOFF, O_Input => I_LC_Con_Present, O_InputDelayOn => DON_LC_Con_Present);
LC_Con_Free_Front(Enable := Enable, I_Input := Inputs.LC_Con_Free_Front, TimeDelayOn := Settings.TimeConFreeFrontDON, TimeDelayOff := Settings.TimeConFreeFrontDOFF, O_Input => I_LC_Con_Free_Front, O_InputDelayOn => DON_LC_Con_Free_front, O_InputDelayOff => DOff_LC_Con_Free_front);
IS_Act_Back_Out(Enable := Enable, I_Input := Inputs.IS_Act_Back_Out, TimeDelayOn := UINT#1, TimeDelayOff := UINT#1, O_Input => I_IS_Act_Back_Out);
IS_Act_Back_In(Enable := Enable, I_Input := Inputs.IS_Act_Back_In, TimeDelayOn := UINT#1, TimeDelayOff := UINT#1, O_Input => I_IS_Act_Back_In);
IS_Act_Front_Out(Enable := Enable, I_Input := Inputs.IS_Act_Front_Out, TimeDelayOn := UINT#1, TimeDelayOff := UINT#1, O_Input => I_IS_Act_Front_Out);
IS_Act_Front_In(Enable := Enable, I_Input := Inputs.IS_Act_Front_In, TimeDelayOn := UINT#1, TimeDelayOff := UINT#1, O_Input => I_IS_Act_Front_In);
IS_Lift_Level(Enable := Enable, I_Input := Inputs.IS_Lift_Level, TimeDelayOn := UINT#1, TimeDelayOff := UINT#1, O_Input => I_IS_Lift_Level);
IS_Con_In_Pos_Back(Enable := Enable, I_Input := Inputs.IS_Con_In_Pos_Back, TimeDelayOn := Settings.TimeConInductiveBackDON, TimeDelayOff := Settings.TimeConInductiveBackDOFF, O_Input => I_IS_Con_In_Pos_Back, O_InputDelayOn => DON_IS_Con_In_Pos_Back, O_InputDelayOff => DOFF_IS_Con_In_Pos_Back);
IS_Con_In_Pos_Front(Enable := Enable, I_Input := Inputs.IS_Con_In_Pos_Front, TimeDelayOn := Settings.TimeConInductiveFrontDON, TimeDelayOff := Settings.TimeConInductiveFrontDOFF, O_Input => I_IS_Con_In_Pos_Front, O_InputDelayOn => DON_IS_Con_In_Pos_Front, O_InputDelayOff => DOFF_IS_Con_In_Pos_Front);

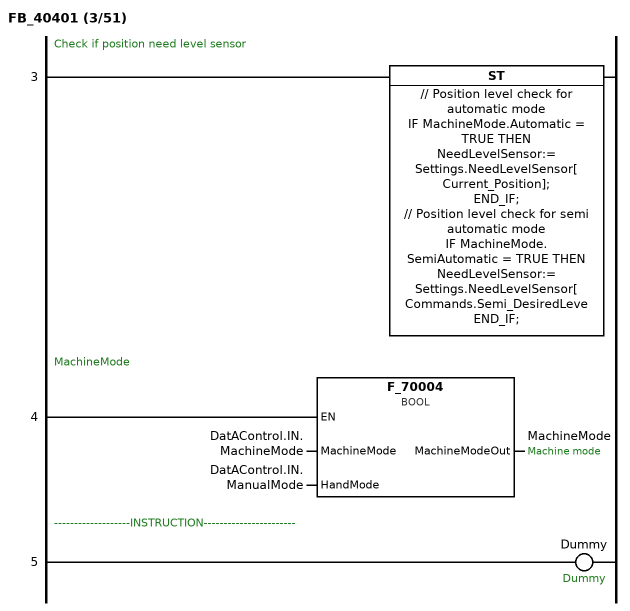
(* Rung 3: Check if position need level sensor *)
// Position level check for automatic mode
IF MachineMode.Automatic = TRUE THEN
	NeedLevelSensor:= Settings.NeedLevelSensor[Current_Position];
END_IF;

// Position level check for semi automatic mode
IF MachineMode.SemiAutomatic = TRUE THEN
	NeedLevelSensor:= Settings.NeedLevelSensor[Commands.Semi_DesiredLevel];
END_IF;
(* Rung 4: MachineMode *)
_t1 := F_70004(MachineMode := DatAControl.IN.MachineMode, HandMode := DatAControl.IN.ManualMode, MachineModeOut => MachineMode);
(* Rung 5: -------------------INSTRUCTION----------------------- *)
Dummy := TRUE;

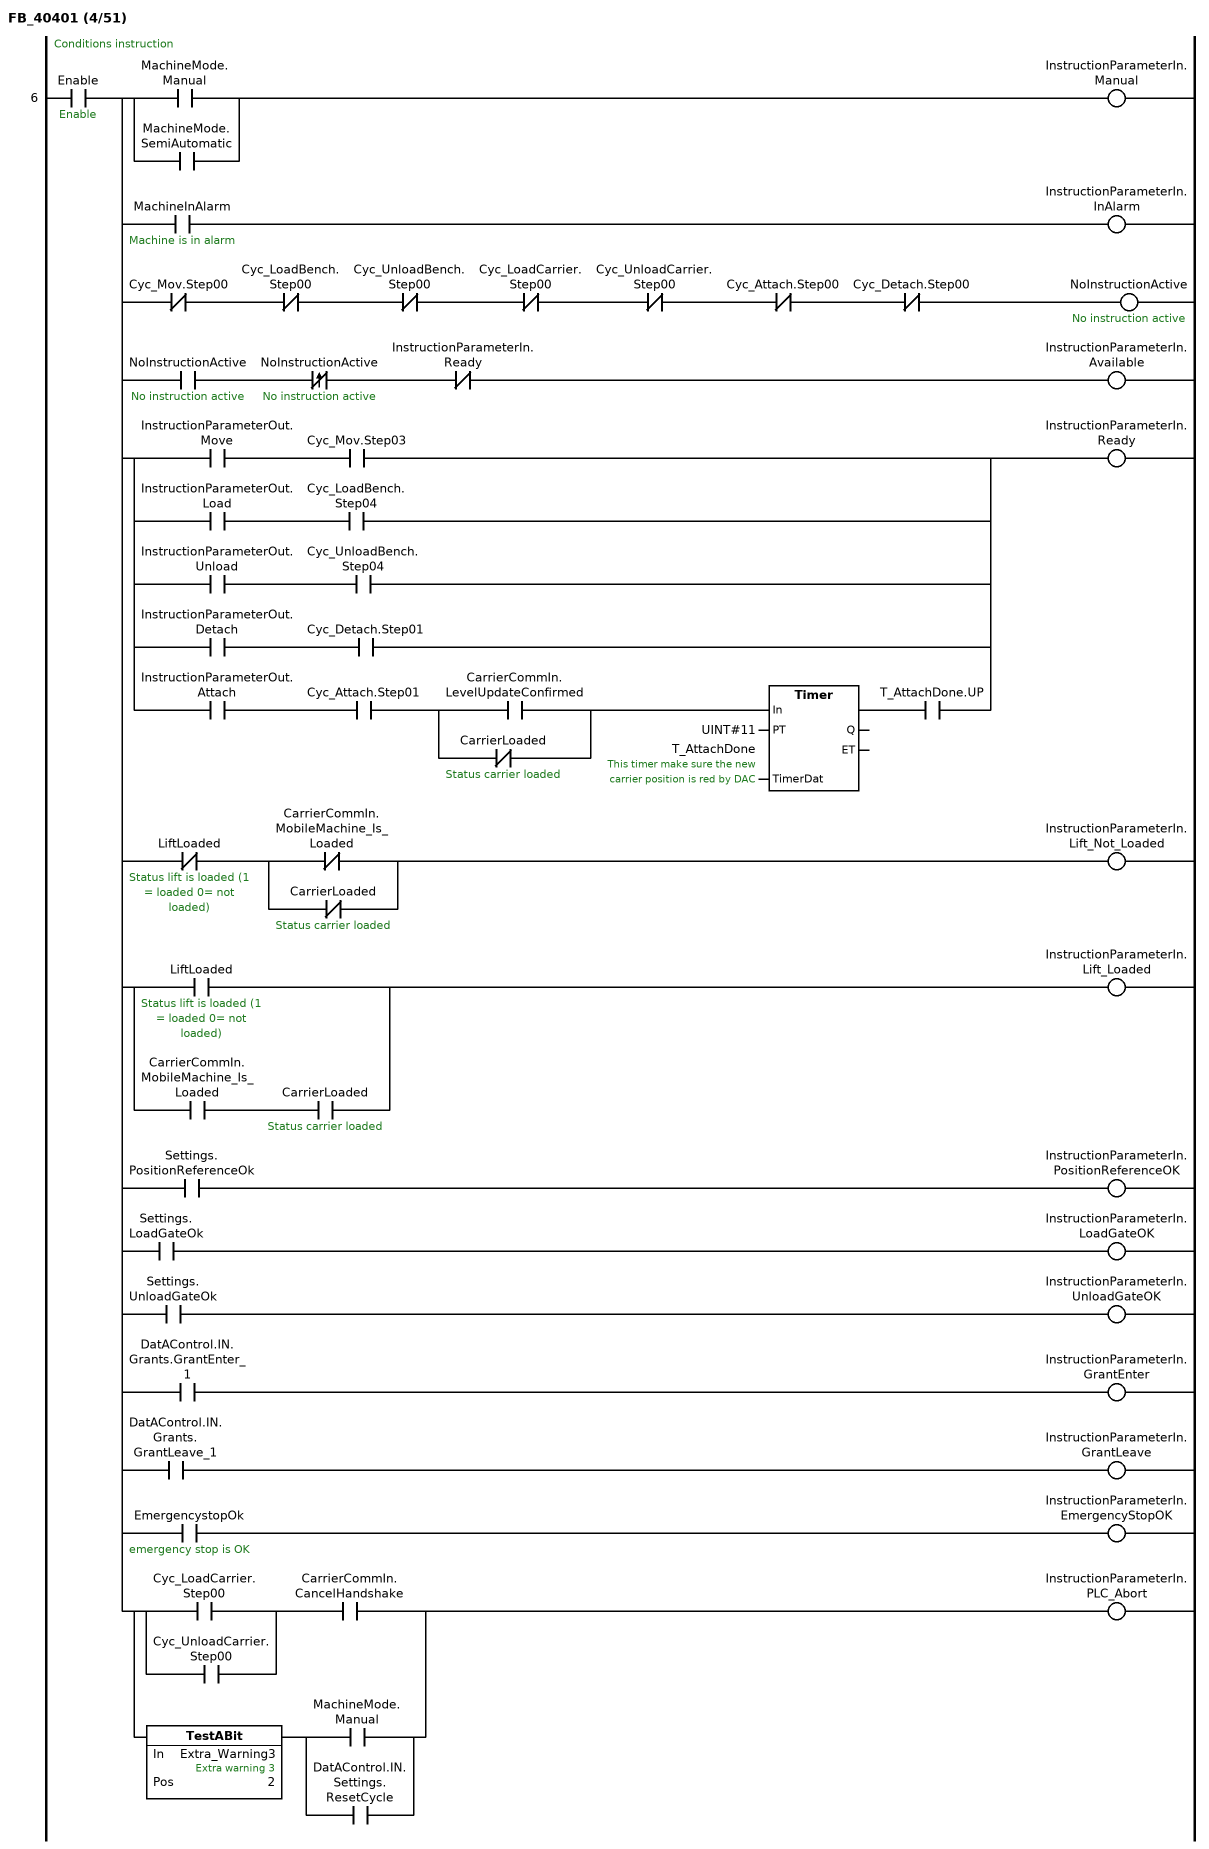
(* Rung 6: Conditions instruction *)
InstructionParameterIn.Manual := Enable AND (MachineMode.Manual OR MachineMode.SemiAutomatic);
InstructionParameterIn.InAlarm := Enable AND MachineInAlarm;
NoInstructionActive := Enable AND NOT Cyc_Mov.Step00 AND NOT Cyc_LoadBench.Step00 AND NOT Cyc_UnloadBench.Step00 AND NOT Cyc_LoadCarrier.Step00 AND NOT Cyc_UnloadCarrier.Step00 AND NOT Cyc_Attach.Step00 AND NOT Cyc_Detach.Step00;
_e2(CLK := NoInstructionActive);
InstructionParameterIn.Available := Enable AND NoInstructionActive AND NOT _e2.Q AND NOT InstructionParameterIn.Ready;
_t3 := Timer(In := Enable AND InstructionParameterOut.Attach AND Cyc_Attach.Step01 AND (CarrierCommIn.LevelUpdateConfirmed OR NOT CarrierLoaded), PT := UINT#11, TimerDat := T_AttachDone);
InstructionParameterIn.Ready := (Enable AND ((InstructionParameterOut.Move AND Cyc_Mov.Step03) OR (InstructionParameterOut.Load AND Cyc_LoadBench.Step04) OR (InstructionParameterOut.Unload AND Cyc_UnloadBench.Step04) OR (InstructionParameterOut.Detach AND Cyc_Detach.Step01))) OR (_t3 AND T_AttachDone.UP);
InstructionParameterIn.Lift_Not_Loaded := Enable AND NOT LiftLoaded AND (NOT CarrierCommIn.MobileMachine_Is_Loaded OR NOT CarrierLoaded);
InstructionParameterIn.Lift_Loaded := Enable AND (LiftLoaded OR (CarrierCommIn.MobileMachine_Is_Loaded AND CarrierLoaded));
InstructionParameterIn.PositionReferenceOK := Enable AND Settings.PositionReferenceOk;
InstructionParameterIn.LoadGateOK := Enable AND Settings.LoadGateOk;
InstructionParameterIn.UnloadGateOK := Enable AND Settings.UnloadGateOk;
InstructionParameterIn.GrantEnter := Enable AND DatAControl.IN.Grants.GrantEnter_1;
InstructionParameterIn.GrantLeave := Enable AND DatAControl.IN.Grants.GrantLeave_1;
InstructionParameterIn.EmergencyStopOK := Enable AND EmergencystopOk;
InstructionParameterIn.PLC_Abort := Enable AND (((Cyc_LoadCarrier.Step00 OR Cyc_UnloadCarrier.Step00) AND CarrierCommIn.CancelHandshake) OR (TestABit(In := Extra_Warning3, Pos := 2) AND (MachineMode.Manual OR DatAControl.IN.Settings.ResetCycle)));

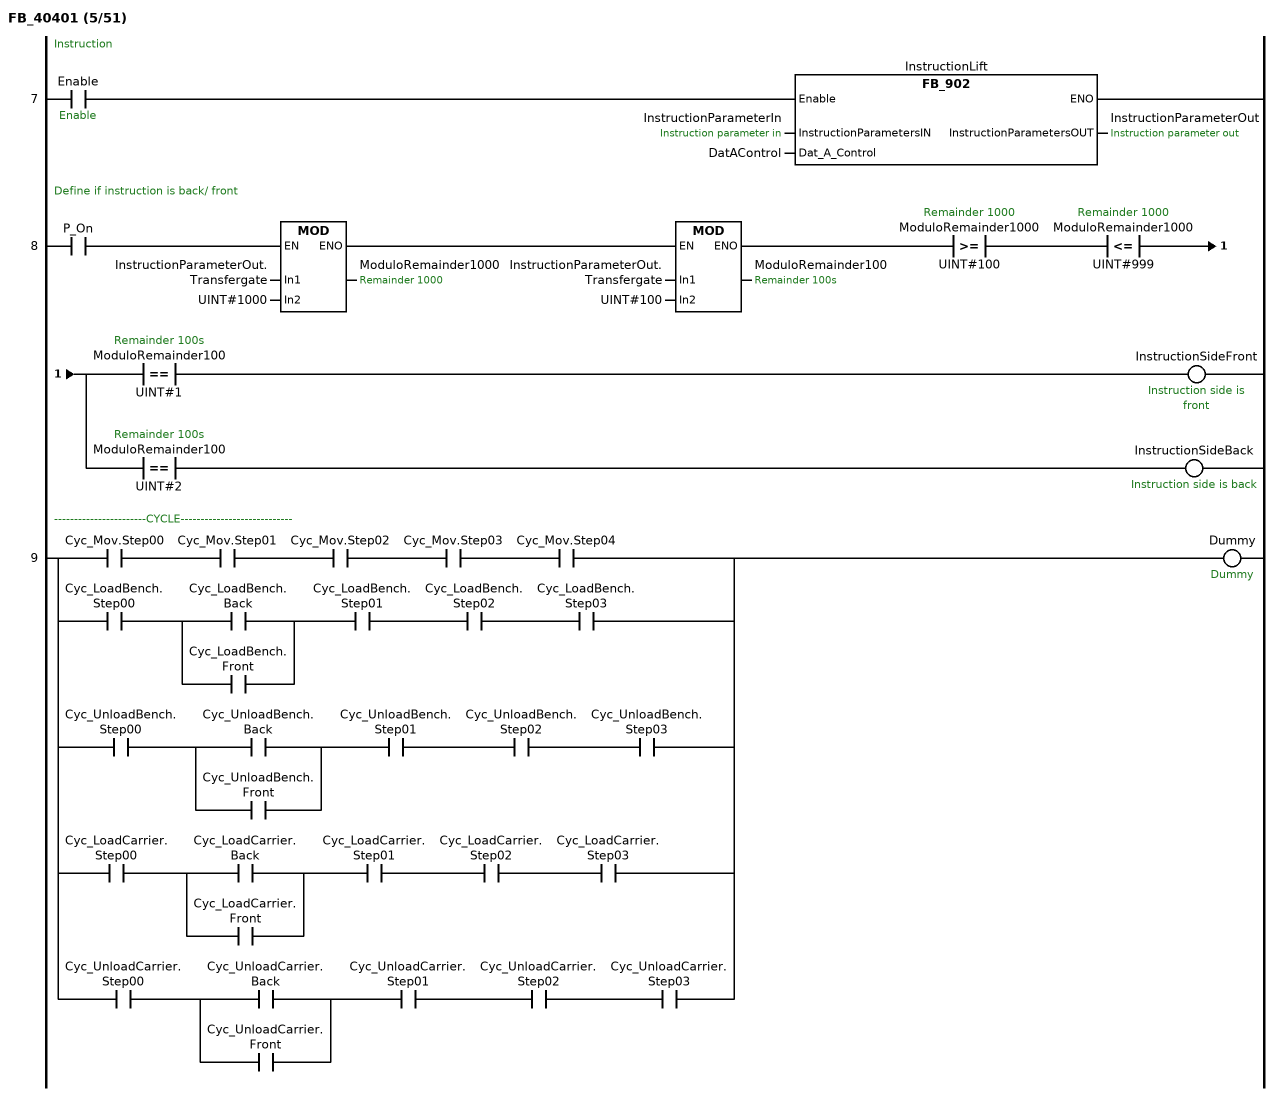
(* Rung 7: Instruction *)
InstructionLift(Enable := Enable, InstructionParametersIN := InstructionParameterIn, Dat_A_Control := DatAControl, InstructionParametersOUT => InstructionParameterOut);
(* Rung 8: Define if instruction is back/ front *)
IF P_On THEN
    ModuloRemainder1000 := InstructionParameterOut.Transfergate MOD UINT#1000;
    ModuloRemainder100 := InstructionParameterOut.Transfergate MOD UINT#100;
END_IF;
_p4 := P_On AND (ModuloRemainder1000 >= UINT#100) AND (ModuloRemainder1000 <= UINT#999);
InstructionSideFront := _p4 AND (ModuloRemainder100 = UINT#1);
InstructionSideBack := _p4 AND (ModuloRemainder100 = UINT#2);
(* Rung 9: -----------------------CYCLE---------------------------- *)
Dummy := (Cyc_Mov.Step00 AND Cyc_Mov.Step01 AND Cyc_Mov.Step02 AND Cyc_Mov.Step03 AND Cyc_Mov.Step04) OR (Cyc_LoadBench.Step00 AND (Cyc_LoadBench.Back OR Cyc_LoadBench.Front) AND Cyc_LoadBench.Step01 AND Cyc_LoadBench.Step02 AND Cyc_LoadBench.Step03) OR (Cyc_UnloadBench.Step00 AND (Cyc_UnloadBench.Back OR Cyc_UnloadBench.Front) AND Cyc_UnloadBench.Step01 AND Cyc_UnloadBench.Step02 AND Cyc_UnloadBench.Step03) OR (Cyc_LoadCarrier.Step00 AND (Cyc_LoadCarrier.Back OR Cyc_LoadCarrier.Front) AND Cyc_LoadCarrier.Step01 AND Cyc_LoadCarrier.Step02 AND Cyc_LoadCarrier.Step03) OR (Cyc_UnloadCarrier.Step00 AND (Cyc_UnloadCarrier.Back OR Cyc_UnloadCarrier.Front) AND Cyc_UnloadCarrier.Step01 AND Cyc_UnloadCarrier.Step02 AND Cyc_UnloadCarrier.Step03);

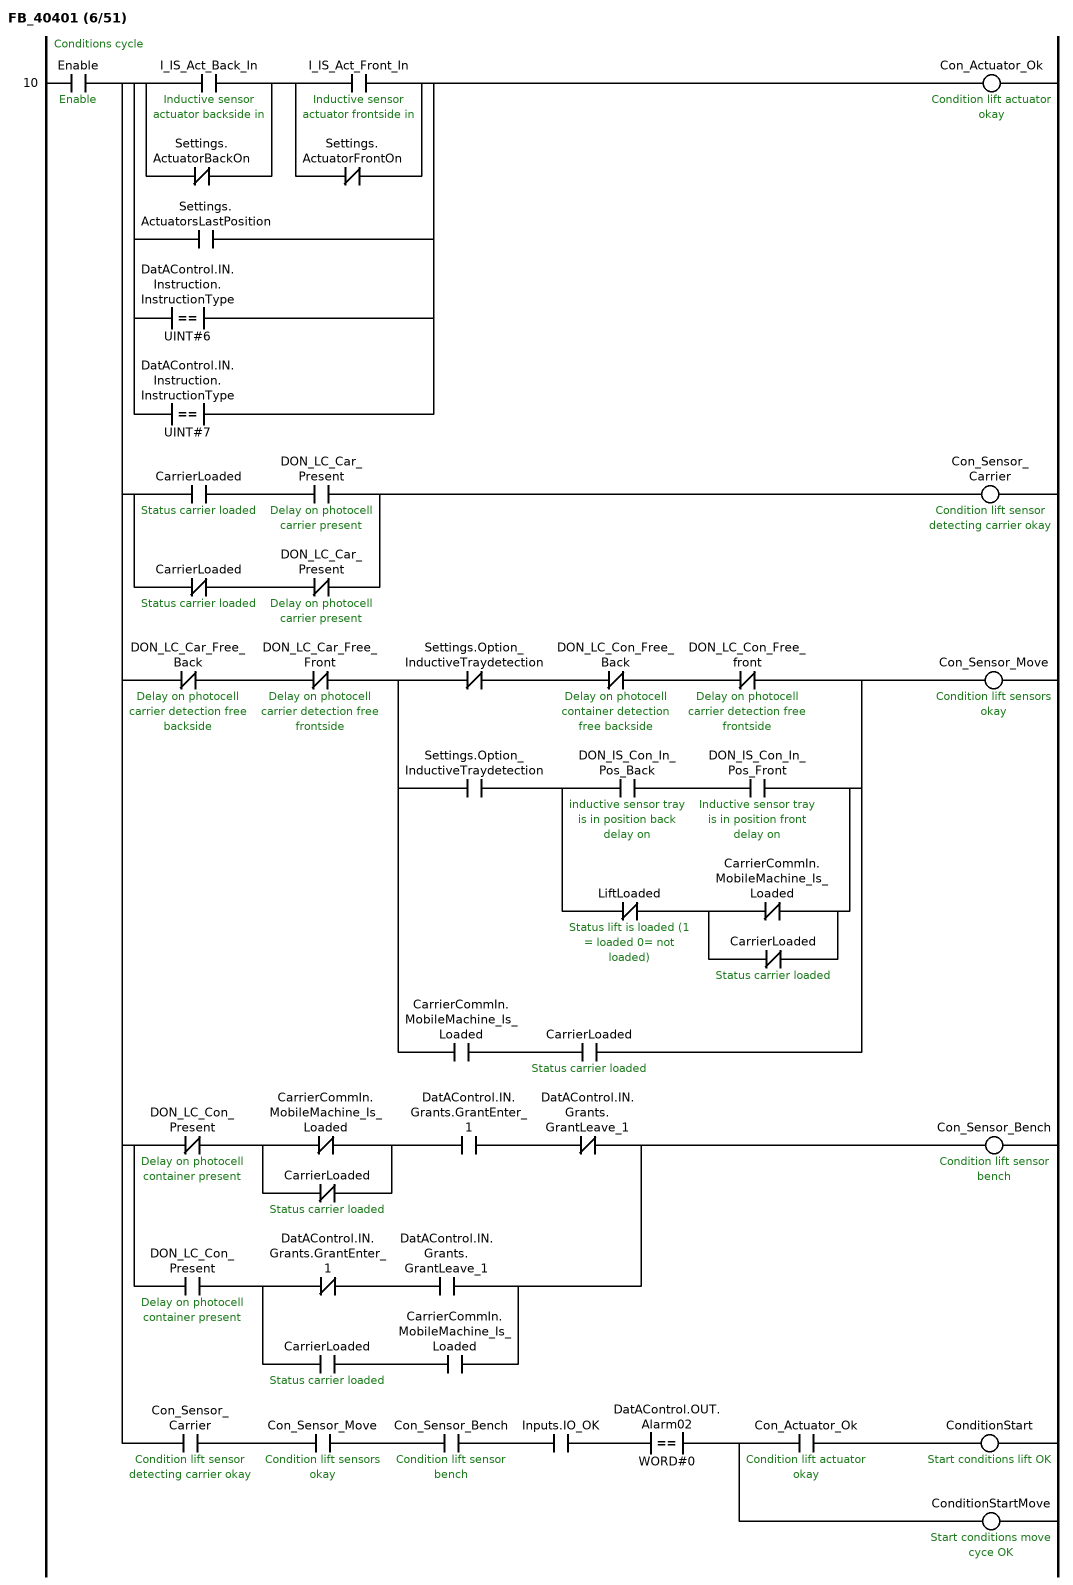
(* Rung 10: Conditions cycle *)
Con_Actuator_Ok := Enable AND (((I_IS_Act_Back_In OR NOT Settings.ActuatorBackOn) AND (I_IS_Act_Front_In OR NOT Settings.ActuatorFrontOn)) OR Settings.ActuatorsLastPosition OR (DatAControl.IN.Instruction.InstructionType = UINT#6) OR (DatAControl.IN.Instruction.InstructionType = UINT#7));
Con_Sensor_Carrier := Enable AND ((CarrierLoaded AND DON_LC_Car_Present) OR (NOT CarrierLoaded AND NOT DON_LC_Car_Present));
Con_Sensor_Move := Enable AND NOT DON_LC_Car_Free_Back AND NOT DON_LC_Car_Free_Front AND ((NOT Settings.Option_InductiveTraydetection AND NOT DON_LC_Con_Free_Back AND NOT DON_LC_Con_Free_front) OR (Settings.Option_InductiveTraydetection AND ((DON_IS_Con_In_Pos_Back AND DON_IS_Con_In_Pos_Front) OR (NOT LiftLoaded AND (NOT CarrierCommIn.MobileMachine_Is_Loaded OR NOT CarrierLoaded)))) OR (CarrierCommIn.MobileMachine_Is_Loaded AND CarrierLoaded));
Con_Sensor_Bench := Enable AND ((NOT DON_LC_Con_Present AND (NOT CarrierCommIn.MobileMachine_Is_Loaded OR NOT CarrierLoaded) AND DatAControl.IN.Grants.GrantEnter_1 AND NOT DatAControl.IN.Grants.GrantLeave_1) OR (DON_LC_Con_Present AND ((NOT DatAControl.IN.Grants.GrantEnter_1 AND DatAControl.IN.Grants.GrantLeave_1) OR (CarrierLoaded AND CarrierCommIn.MobileMachine_Is_Loaded))));
_p5 := Enable AND Con_Sensor_Carrier AND Con_Sensor_Move AND Con_Sensor_Bench AND Inputs.IO_OK AND (DatAControl.OUT.Alarm02 = WORD#0);
ConditionStart := _p5 AND Con_Actuator_Ok;
ConditionStartMove := _p5;

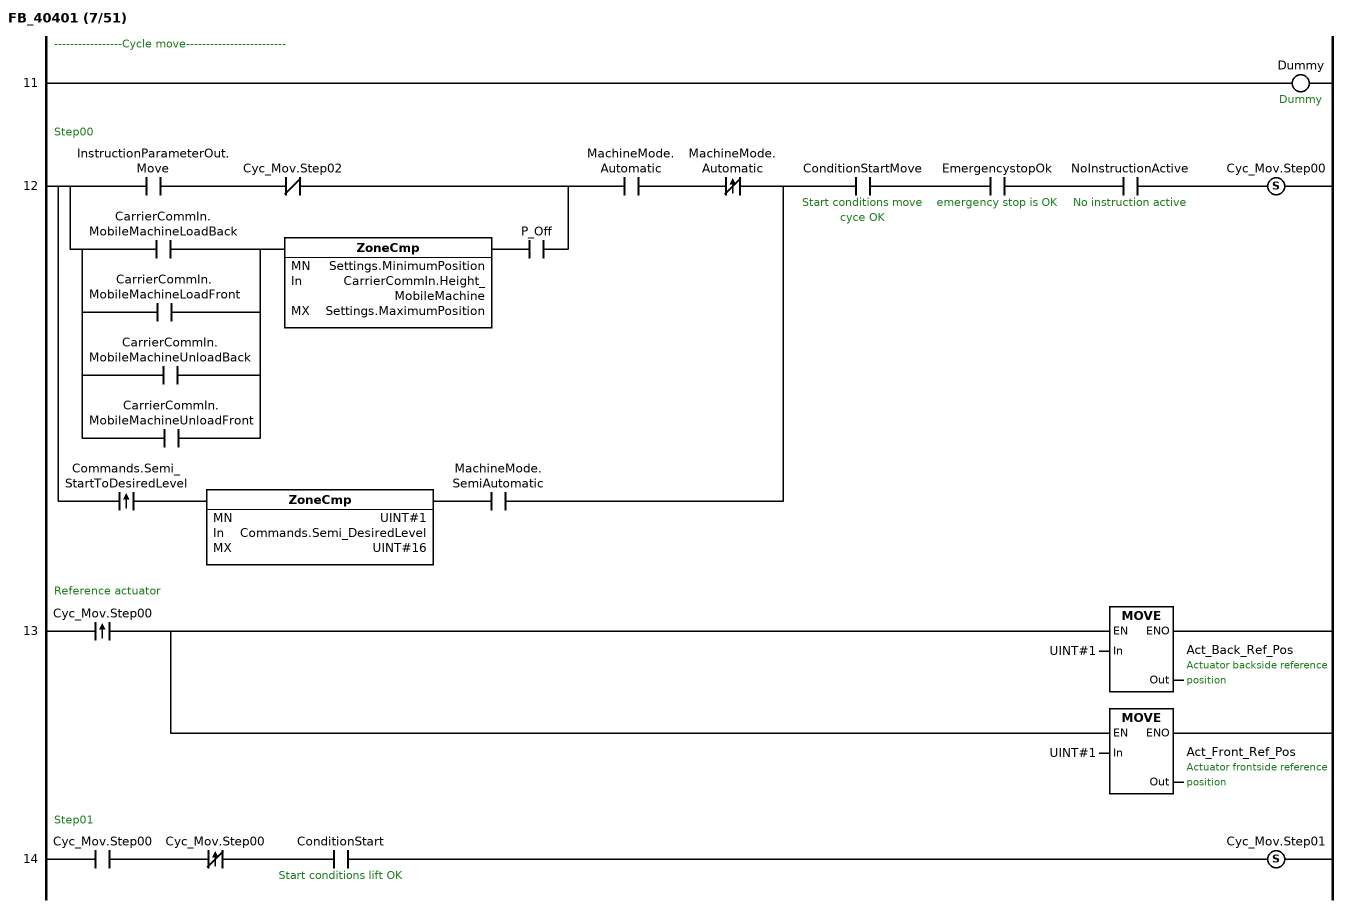
(* Rung 11: -----------------Cycle move------------------------- *)
Dummy := TRUE;
(* Rung 12: Step00 *)
_e6(CLK := MachineMode.Automatic);
_e7(CLK := Commands.Semi_StartToDesiredLevel);
IF ((((InstructionParameterOut.Move AND NOT Cyc_Mov.Step02) OR ((CarrierCommIn.MobileMachineLoadBack OR CarrierCommIn.MobileMachineLoadFront OR CarrierCommIn.MobileMachineUnloadBack OR CarrierCommIn.MobileMachineUnloadFront) AND ZoneCmp(MN := Settings.MinimumPosition, In := CarrierCommIn.Height_MobileMachine, MX := Settings.MaximumPosition) AND P_Off)) AND MachineMode.Automatic AND NOT _e6.Q) OR (_e7.Q AND ZoneCmp(MN := UINT#1, In := Commands.Semi_DesiredLevel, MX := UINT#16) AND MachineMode.SemiAutomatic)) AND ConditionStartMove AND EmergencystopOk AND NoInstructionActive THEN
    Cyc_Mov.Step00 := TRUE;
END_IF;
(* Rung 13: Reference actuator *)
_e8(CLK := Cyc_Mov.Step00);
IF _e8.Q THEN
    Act_Back_Ref_Pos := UINT#1;
    Act_Front_Ref_Pos := UINT#1;
END_IF;
(* Rung 14: Step01 *)
_e9(CLK := Cyc_Mov.Step00);
IF Cyc_Mov.Step00 AND NOT _e9.Q AND ConditionStart THEN Cyc_Mov.Step01 := TRUE; END_IF;

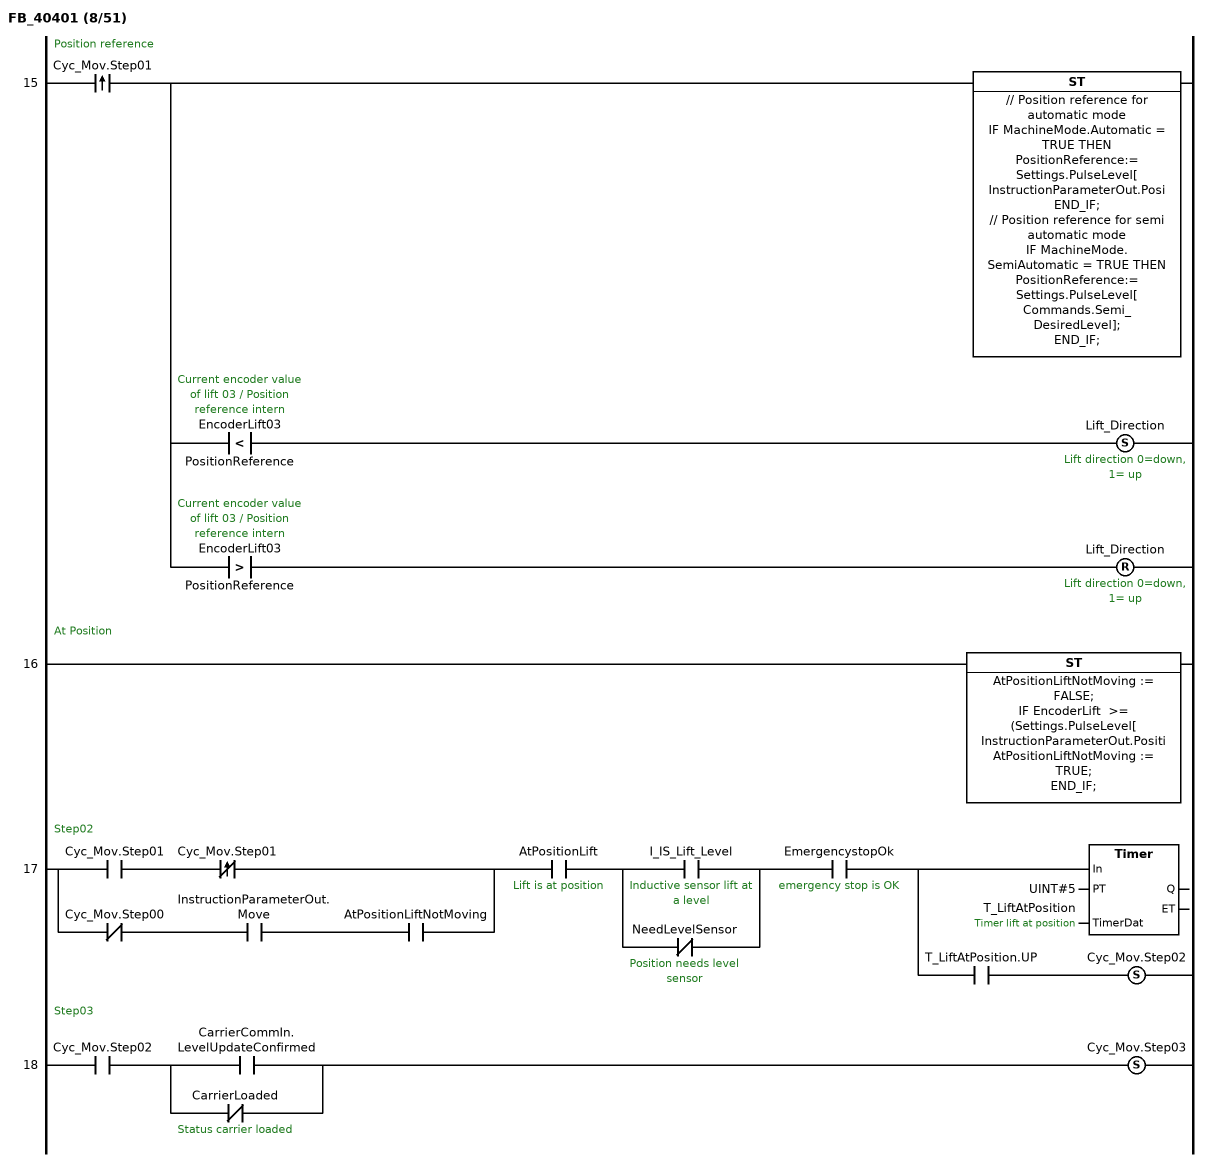
(* Rung 15: Position reference *)
_e10(CLK := Cyc_Mov.Step01);
IF _e10.Q THEN
    // Position reference for automatic mode
    IF MachineMode.Automatic = TRUE THEN
    	PositionReference:= Settings.PulseLevel[InstructionParameterOut.Position];
    END_IF;
    
    // Position reference for semi automatic mode
    IF MachineMode.SemiAutomatic = TRUE THEN
    	PositionReference:= Settings.PulseLevel[Commands.Semi_DesiredLevel];
    END_IF;
END_IF;
IF _e10.Q AND (EncoderLift03 < PositionReference) THEN Lift_Direction := TRUE; END_IF;
IF _e10.Q AND (EncoderLift03 > PositionReference) THEN Lift_Direction := FALSE; END_IF;
(* Rung 16: At Position *)
AtPositionLiftNotMoving := FALSE;

IF EncoderLift  >= (Settings.PulseLevel[InstructionParameterOut.Position] - Settings.Tolerance_At_Position) AND EncoderLift <= (Settings.PulseLevel[InstructionParameterOut.Position] + Settings.Tolerance_At_Position) THEN
	AtPositionLiftNotMoving := TRUE;
END_IF;
(* Rung 17: Step02 *)
_e11(CLK := Cyc_Mov.Step01);
_p12 := ((Cyc_Mov.Step01 AND NOT _e11.Q) OR (NOT Cyc_Mov.Step00 AND InstructionParameterOut.Move AND AtPositionLiftNotMoving)) AND AtPositionLift AND (I_IS_Lift_Level OR NOT NeedLevelSensor) AND EmergencystopOk;
_t13 := Timer(In := _p12, PT := UINT#5, TimerDat := T_LiftAtPosition);
IF _p12 AND T_LiftAtPosition.UP THEN Cyc_Mov.Step02 := TRUE; END_IF;
(* Rung 18: Step03 *)
IF Cyc_Mov.Step02 AND (CarrierCommIn.LevelUpdateConfirmed OR NOT CarrierLoaded) THEN
    Cyc_Mov.Step03 := TRUE;
END_IF;

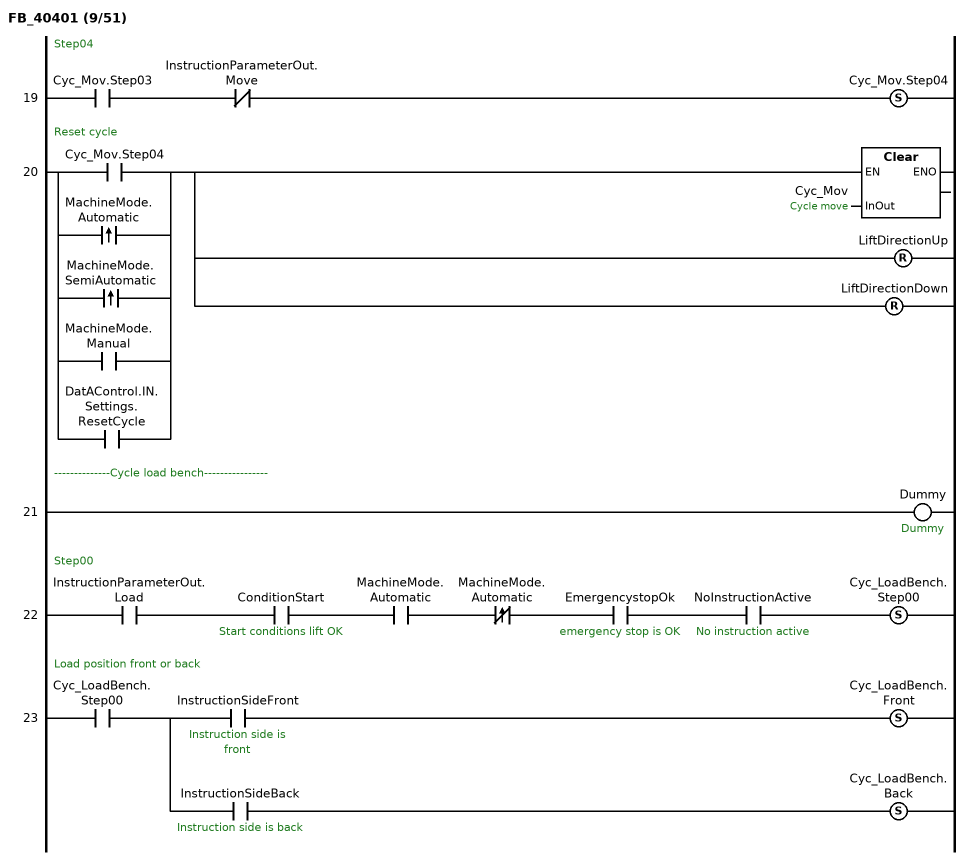
(* Rung 19: Step04 *)
IF Cyc_Mov.Step03 AND NOT InstructionParameterOut.Move THEN Cyc_Mov.Step04 := TRUE; END_IF;
(* Rung 20: Reset cycle *)
_e14(CLK := MachineMode.Automatic);
_e15(CLK := MachineMode.SemiAutomatic);
_p16 := Cyc_Mov.Step04 OR _e14.Q OR _e15.Q OR MachineMode.Manual OR DatAControl.IN.Settings.ResetCycle;
IF _p16 THEN
    Clear(InOut := Cyc_Mov);
    LiftDirectionUp := FALSE;
    LiftDirectionDown := FALSE;
END_IF;
(* Rung 21: --------------Cycle load bench---------------- *)
Dummy := TRUE;
(* Rung 22: Step00 *)
_e17(CLK := MachineMode.Automatic);
IF InstructionParameterOut.Load AND ConditionStart AND MachineMode.Automatic AND NOT _e17.Q AND EmergencystopOk AND NoInstructionActive THEN
    Cyc_LoadBench.Step00 := TRUE;
END_IF;
(* Rung 23: Load position front or back *)
_p18 := Cyc_LoadBench.Step00;
IF Cyc_LoadBench.Step00 AND InstructionSideFront THEN Cyc_LoadBench.Front := TRUE; END_IF;
IF _p18 AND InstructionSideBack THEN Cyc_LoadBench.Back := TRUE; END_IF;

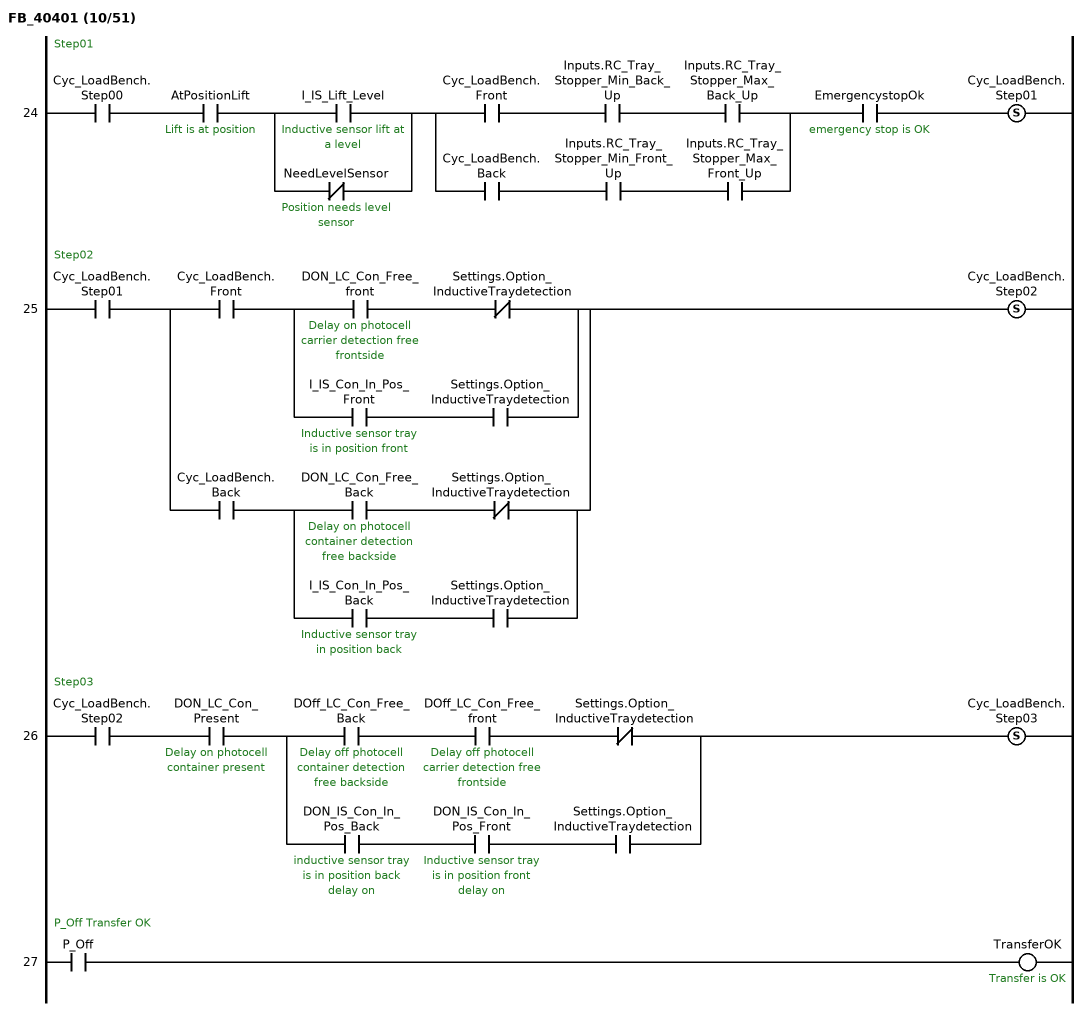
(* Rung 24: Step01 *)
IF Cyc_LoadBench.Step00 AND AtPositionLift AND (I_IS_Lift_Level OR NOT NeedLevelSensor) AND ((Cyc_LoadBench.Front AND Inputs.RC_Tray_Stopper_Min_Back_Up AND Inputs.RC_Tray_Stopper_Max_Back_Up) OR (Cyc_LoadBench.Back AND Inputs.RC_Tray_Stopper_Min_Front_Up AND Inputs.RC_Tray_Stopper_Max_Front_Up)) AND EmergencystopOk THEN
    Cyc_LoadBench.Step01 := TRUE;
END_IF;
(* Rung 25: Step02 *)
IF Cyc_LoadBench.Step01 AND ((Cyc_LoadBench.Front AND ((DON_LC_Con_Free_front AND NOT Settings.Option_InductiveTraydetection) OR (I_IS_Con_In_Pos_Front AND Settings.Option_InductiveTraydetection))) OR (Cyc_LoadBench.Back AND ((DON_LC_Con_Free_Back AND NOT Settings.Option_InductiveTraydetection) OR (I_IS_Con_In_Pos_Back AND Settings.Option_InductiveTraydetection)))) THEN
    Cyc_LoadBench.Step02 := TRUE;
END_IF;
(* Rung 26: Step03 *)
IF Cyc_LoadBench.Step02 AND DON_LC_Con_Present AND ((DOff_LC_Con_Free_Back AND DOff_LC_Con_Free_front AND NOT Settings.Option_InductiveTraydetection) OR (DON_IS_Con_In_Pos_Back AND DON_IS_Con_In_Pos_Front AND Settings.Option_InductiveTraydetection)) THEN
    Cyc_LoadBench.Step03 := TRUE;
END_IF;
(* Rung 27: P_Off Transfer OK *)
TransferOK := P_Off;

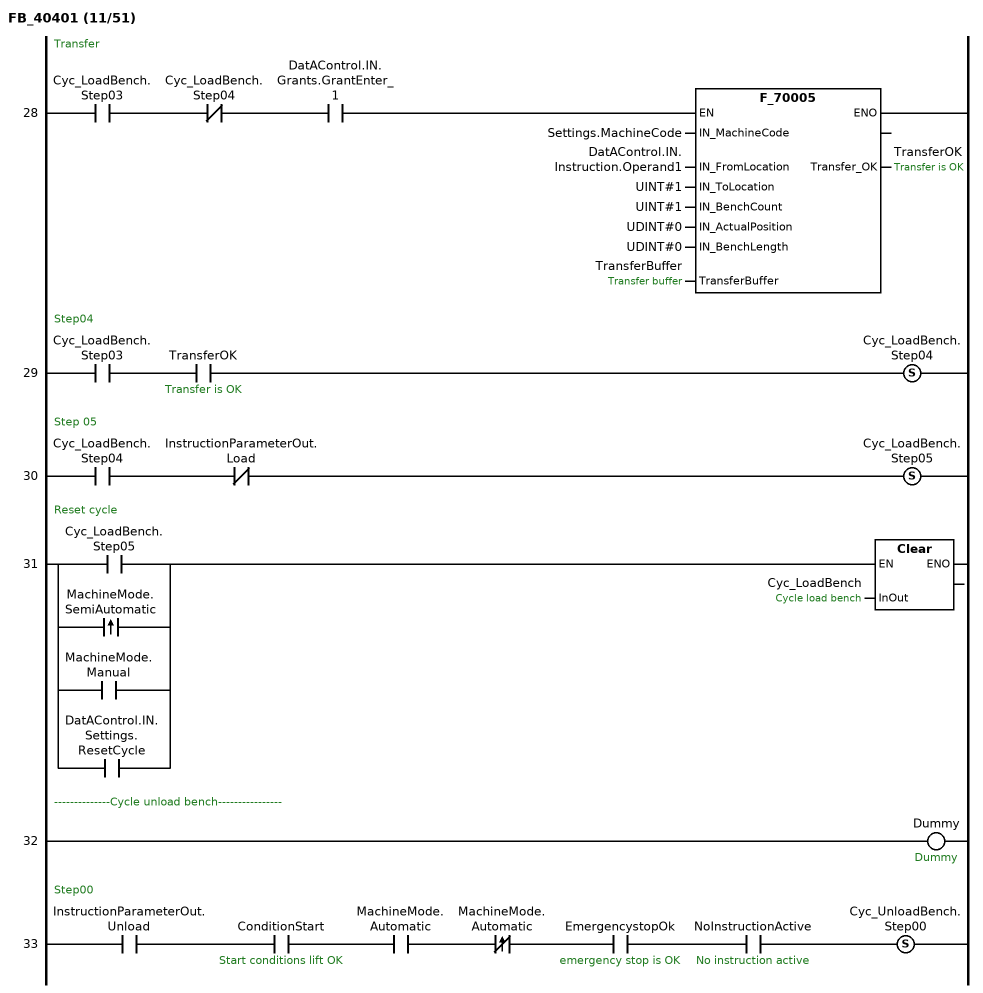
(* Rung 28: Transfer *)
IF Cyc_LoadBench.Step03 AND NOT Cyc_LoadBench.Step04 AND DatAControl.IN.Grants.GrantEnter_1 THEN
    F_70005(IN_MachineCode := Settings.MachineCode, IN_FromLocation := DatAControl.IN.Instruction.Operand1, IN_ToLocation := UINT#1, IN_BenchCount := UINT#1, IN_ActualPosition := UDINT#0, IN_BenchLength := UDINT#0, TransferBuffer := TransferBuffer, Transfer_OK => TransferOK);
END_IF;
(* Rung 29: Step04 *)
IF Cyc_LoadBench.Step03 AND TransferOK THEN Cyc_LoadBench.Step04 := TRUE; END_IF;
(* Rung 30: Step 05 *)
IF Cyc_LoadBench.Step04 AND NOT InstructionParameterOut.Load THEN Cyc_LoadBench.Step05 := TRUE; END_IF;
(* Rung 31: Reset cycle *)
_e19(CLK := MachineMode.SemiAutomatic);
IF Cyc_LoadBench.Step05 OR _e19.Q OR MachineMode.Manual OR DatAControl.IN.Settings.ResetCycle THEN
    Clear(InOut := Cyc_LoadBench);
END_IF;
(* Rung 32: --------------Cycle unload bench---------------- *)
Dummy := TRUE;
(* Rung 33: Step00 *)
_e20(CLK := MachineMode.Automatic);
IF InstructionParameterOut.Unload AND ConditionStart AND MachineMode.Automatic AND NOT _e20.Q AND EmergencystopOk AND NoInstructionActive THEN
    Cyc_UnloadBench.Step00 := TRUE;
END_IF;

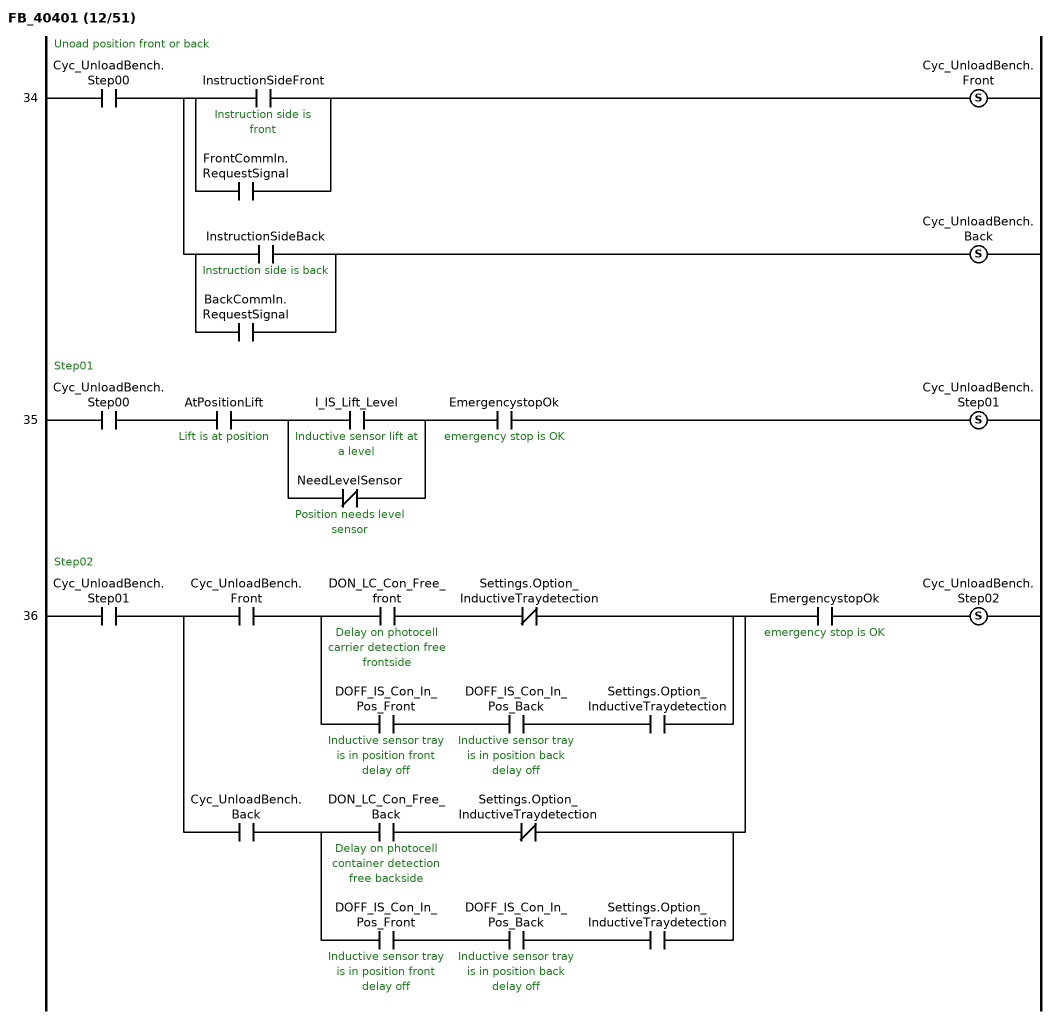
(* Rung 34: Unoad position front or back *)
_p21 := Cyc_UnloadBench.Step00;
IF Cyc_UnloadBench.Step00 AND (InstructionSideFront OR FrontCommIn.RequestSignal) THEN
    Cyc_UnloadBench.Front := TRUE;
END_IF;
IF _p21 AND (InstructionSideBack OR BackCommIn.RequestSignal) THEN Cyc_UnloadBench.Back := TRUE; END_IF;
(* Rung 35: Step01 *)
IF Cyc_UnloadBench.Step00 AND AtPositionLift AND (I_IS_Lift_Level OR NOT NeedLevelSensor) AND EmergencystopOk THEN
    Cyc_UnloadBench.Step01 := TRUE;
END_IF;
(* Rung 36: Step02 *)
IF Cyc_UnloadBench.Step01 AND ((Cyc_UnloadBench.Front AND ((DON_LC_Con_Free_front AND NOT Settings.Option_InductiveTraydetection) OR (DOFF_IS_Con_In_Pos_Front AND DOFF_IS_Con_In_Pos_Back AND Settings.Option_InductiveTraydetection))) OR (Cyc_UnloadBench.Back AND ((DON_LC_Con_Free_Back AND NOT Settings.Option_InductiveTraydetection) OR (DOFF_IS_Con_In_Pos_Front AND DOFF_IS_Con_In_Pos_Back AND Settings.Option_InductiveTraydetection)))) AND EmergencystopOk THEN
    Cyc_UnloadBench.Step02 := TRUE;
END_IF;

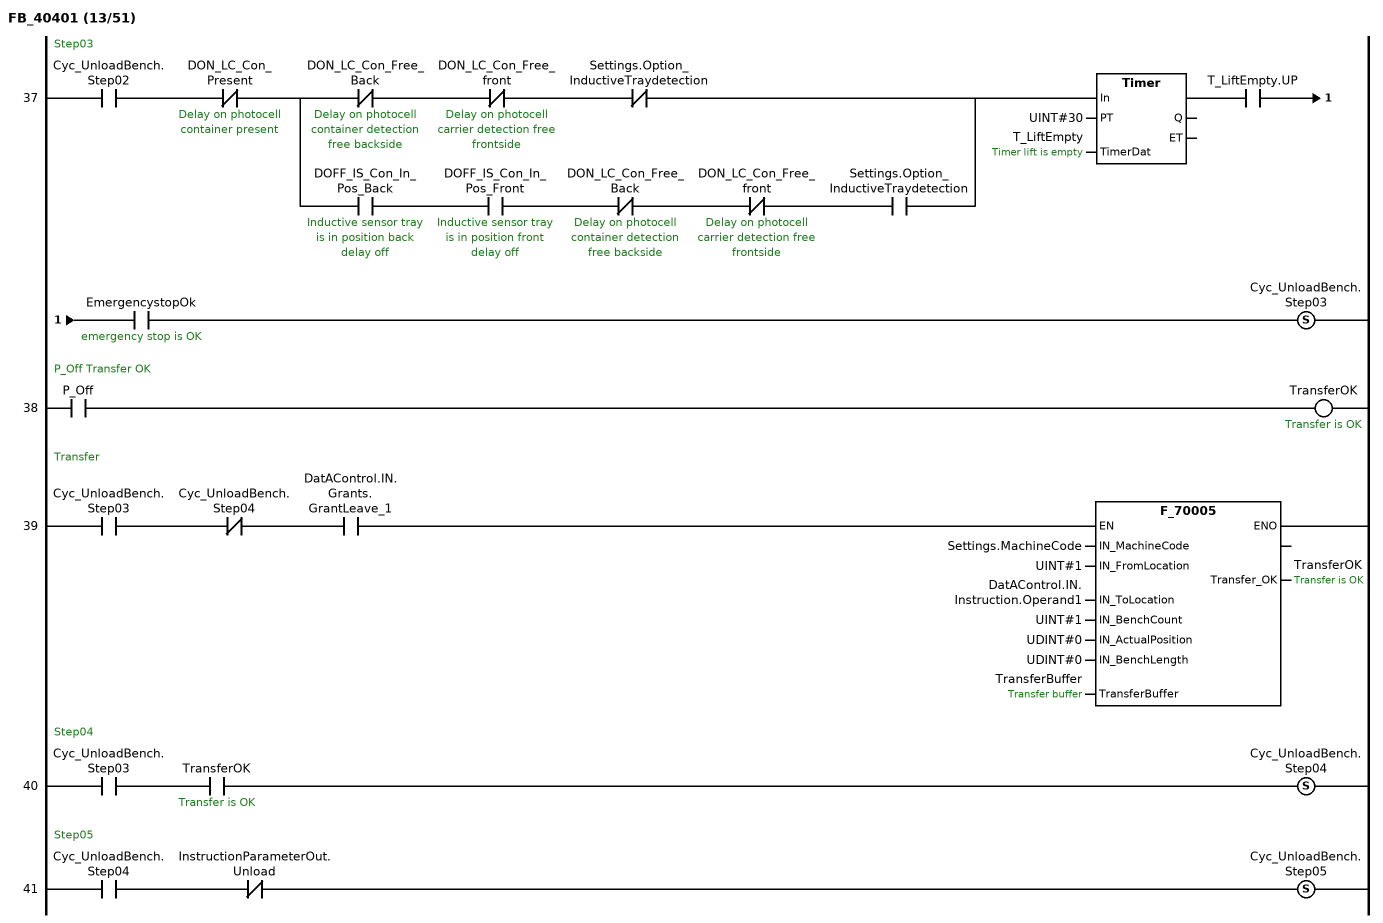
(* Rung 37: Step03 *)
_t22 := Timer(In := Cyc_UnloadBench.Step02 AND NOT DON_LC_Con_Present AND ((NOT DON_LC_Con_Free_Back AND NOT DON_LC_Con_Free_front AND NOT Settings.Option_InductiveTraydetection) OR (DOFF_IS_Con_In_Pos_Back AND DOFF_IS_Con_In_Pos_Front AND NOT DON_LC_Con_Free_Back AND NOT DON_LC_Con_Free_front AND Settings.Option_InductiveTraydetection)), PT := UINT#30, TimerDat := T_LiftEmpty);
IF _t22 AND T_LiftEmpty.UP AND EmergencystopOk THEN Cyc_UnloadBench.Step03 := TRUE; END_IF;
(* Rung 38: P_Off Transfer OK *)
TransferOK := P_Off;
(* Rung 39: Transfer *)
IF Cyc_UnloadBench.Step03 AND NOT Cyc_UnloadBench.Step04 AND DatAControl.IN.Grants.GrantLeave_1 THEN
    F_70005(IN_MachineCode := Settings.MachineCode, IN_FromLocation := UINT#1, IN_ToLocation := DatAControl.IN.Instruction.Operand1, IN_BenchCount := UINT#1, IN_ActualPosition := UDINT#0, IN_BenchLength := UDINT#0, TransferBuffer := TransferBuffer, Transfer_OK => TransferOK);
END_IF;
(* Rung 40: Step04 *)
IF Cyc_UnloadBench.Step03 AND TransferOK THEN Cyc_UnloadBench.Step04 := TRUE; END_IF;
(* Rung 41: Step05 *)
IF Cyc_UnloadBench.Step04 AND NOT InstructionParameterOut.Unload THEN
    Cyc_UnloadBench.Step05 := TRUE;
END_IF;

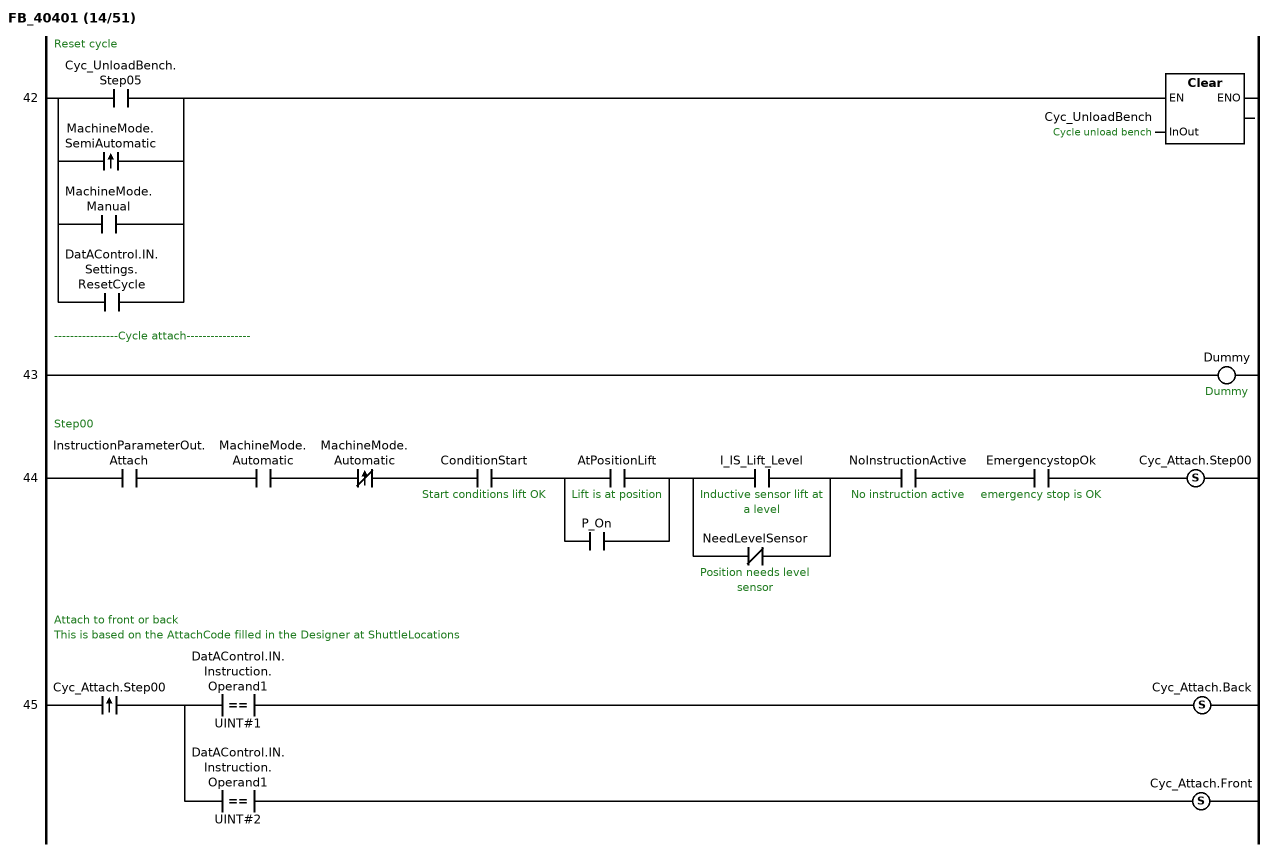
(* Rung 42: Reset cycle *)
_e23(CLK := MachineMode.SemiAutomatic);
IF Cyc_UnloadBench.Step05 OR _e23.Q OR MachineMode.Manual OR DatAControl.IN.Settings.ResetCycle THEN
    Clear(InOut := Cyc_UnloadBench);
END_IF;
(* Rung 43: ----------------Cycle attach---------------- *)
Dummy := TRUE;
(* Rung 44: Step00 *)
_e24(CLK := MachineMode.Automatic);
IF InstructionParameterOut.Attach AND MachineMode.Automatic AND NOT _e24.Q AND ConditionStart AND (AtPositionLift OR P_On) AND (I_IS_Lift_Level OR NOT NeedLevelSensor) AND NoInstructionActive AND EmergencystopOk THEN
    Cyc_Attach.Step00 := TRUE;
END_IF;
(* Rung 45: Attach to front or back / This is based on the AttachCode filled in the Designer at ShuttleLocations *)
_e25(CLK := Cyc_Attach.Step00);
IF _e25.Q AND (DatAControl.IN.Instruction.Operand1 = UINT#1) THEN Cyc_Attach.Back := TRUE; END_IF;
IF _e25.Q AND (DatAControl.IN.Instruction.Operand1 = UINT#2) THEN Cyc_Attach.Front := TRUE; END_IF;

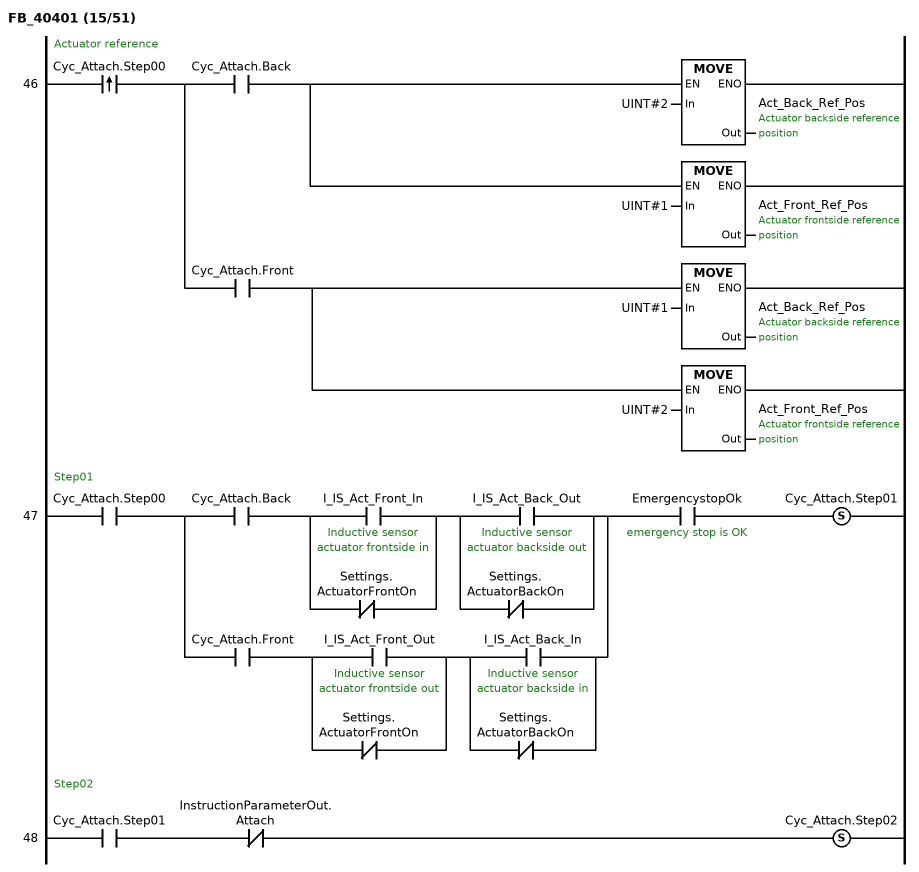
(* Rung 46: Actuator reference *)
_e26(CLK := Cyc_Attach.Step00);
IF _e26.Q AND Cyc_Attach.Back THEN
    Act_Back_Ref_Pos := UINT#2;
    Act_Front_Ref_Pos := UINT#1;
END_IF;
IF _e26.Q AND Cyc_Attach.Front THEN
    Act_Back_Ref_Pos := UINT#1;
    Act_Front_Ref_Pos := UINT#2;
END_IF;
(* Rung 47: Step01 *)
IF Cyc_Attach.Step00 AND ((Cyc_Attach.Back AND (I_IS_Act_Front_In OR NOT Settings.ActuatorFrontOn) AND (I_IS_Act_Back_Out OR NOT Settings.ActuatorBackOn)) OR (Cyc_Attach.Front AND (I_IS_Act_Front_Out OR NOT Settings.ActuatorFrontOn) AND (I_IS_Act_Back_In OR NOT Settings.ActuatorBackOn))) AND EmergencystopOk THEN
    Cyc_Attach.Step01 := TRUE;
END_IF;
(* Rung 48: Step02 *)
IF Cyc_Attach.Step01 AND NOT InstructionParameterOut.Attach THEN Cyc_Attach.Step02 := TRUE; END_IF;

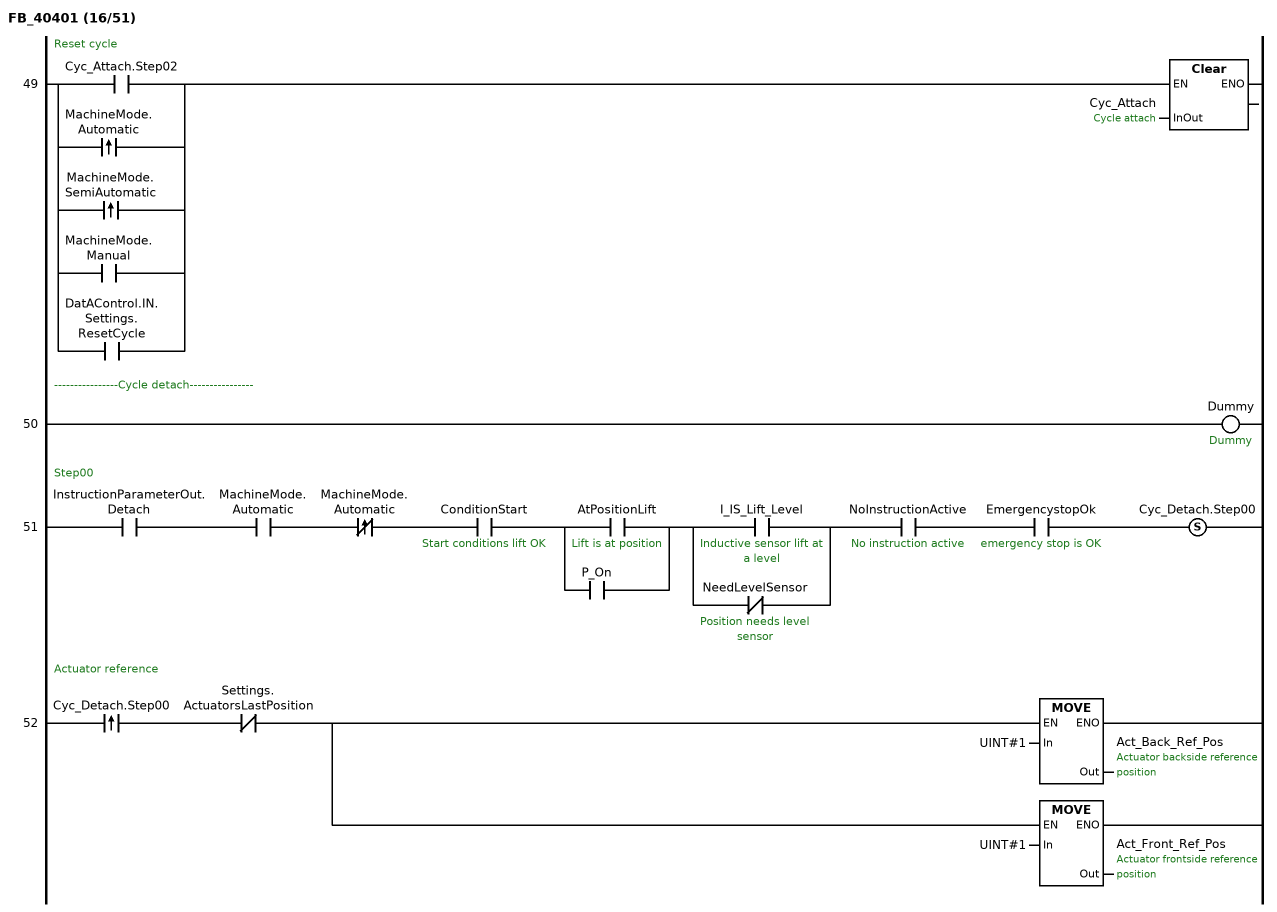
(* Rung 49: Reset cycle *)
_e27(CLK := MachineMode.Automatic);
_e28(CLK := MachineMode.SemiAutomatic);
IF Cyc_Attach.Step02 OR _e27.Q OR _e28.Q OR MachineMode.Manual OR DatAControl.IN.Settings.ResetCycle THEN
    Clear(InOut := Cyc_Attach);
END_IF;
(* Rung 50: ----------------Cycle detach---------------- *)
Dummy := TRUE;
(* Rung 51: Step00 *)
_e29(CLK := MachineMode.Automatic);
IF InstructionParameterOut.Detach AND MachineMode.Automatic AND NOT _e29.Q AND ConditionStart AND (AtPositionLift OR P_On) AND (I_IS_Lift_Level OR NOT NeedLevelSensor) AND NoInstructionActive AND EmergencystopOk THEN
    Cyc_Detach.Step00 := TRUE;
END_IF;
(* Rung 52: Actuator reference *)
_e30(CLK := Cyc_Detach.Step00);
IF _e30.Q AND NOT Settings.ActuatorsLastPosition THEN
    Act_Back_Ref_Pos := UINT#1;
    Act_Front_Ref_Pos := UINT#1;
END_IF;

